NETWORK
TITLE = ---- Final
/////////////////////////////////////////////////////////////////////////
/////////////////////////////////////////////////////////////////////////
/////////////////////////////////////////////////////////////////////////
// Se acabo el evento
Final_EventoRecibido_RETI:NOP   0;
      L     #P_Eventos;  // Recupero por donde voy en la lista de eventos
      LAR2;  // Regreso a buscar el siguiente evento
      JU    FinBucle_EventosRecibidos;



NETWORK
TITLE = Guardar Datos - Evento BORR - Borrar la UT
// Analisis del evento
//   - Inicializa variables de los atributos del Evento
//   - Buscar Atributos o Final del Evento
//   - Guardar datos del Evento
// Analisis de los atributos del Evento
//   - Mirar que atributo del Evento es
//   - Distribuir a recoger los datos del Evento
//   - Recoger el Atributo McKey
//   - Recoger el Atributo MesaActual
GuardarDatos_EventoRecibido_BORR:NOP   0;

/////////////////////////////////////////////////////////////////////////
/////////////////////////////////////////////////////////////////////////
/////////////////////////////////////////////////////////////////////////
// --- Guardar Datos del Evento Recibido


/////////////////////////////////////////////////////////////////////////
/////////////////////////////////////////////////////////////////////////
/////////////////////////////////////////////////////////////////////////
// --- Control de Mesa Recibida
      L     #AtributosDeUTs.MesaActual;
      L     0;
      ==I;
      JC    FinControlMesa_EventoRecibido_BORR;

      L     #AtributosDeUTs.MesaActual;  // Ver que mesa es
      L     "CTE_OffsetMesa";
      -I;
      T     #VarTempUTs.MesaActual;

      L     #VarTempUTs.MesaActual;  // Comprobar el numero de mesa
      L     1;  // No menor de 1
      <I;  // No es correcto
      JC    Final_EventoRecibido_BORR;
      L     #VarTempUTs.MesaActual;
      L     "CTE_MaxMesas";  // No mayor que el parametro
      >I;  // No es correcto
      JC    Final_EventoRecibido_BORR;

/////////////////////////////////////////////////////////////////////////
FinControlMesa_EventoRecibido_BORR:NOP   0;



NETWORK
TITLE = ---- Accion del Evento --> Distribucion
/////////////////////////////////////////////////////////////////////////
/////////////////////////////////////////////////////////////////////////
/////////////////////////////////////////////////////////////////////////
// --- Distribucion

      L     0;  // Borrar UT en Particular
      L     #AtributosDeUTs.Mckey;
      <>D;
      JC    BorrarUT_EventoRecibido_BORR;

      L     0;  // Borrar UTs de la Mesa
      L     #AtributosDeUTs.MesaActual;
      <>I;
      JC    BorrarUTsDeMesa_EventoRecibido_BORR;

/////////////////////////////////////////////////////////////////////////
// --- Defecto --> Borrar todas las UTs
      JU    BorrarTodasLasUTs_EventoRecibido_BORR;



NETWORK
TITLE = ---- Accion del Evento --> Borrar UT
/////////////////////////////////////////////////////////////////////////
/////////////////////////////////////////////////////////////////////////
/////////////////////////////////////////////////////////////////////////
// --- Borrar una UT en particular
BorrarUT_EventoRecibido_BORR:NOP   0;
      L     #AtributosDeUTs.MesaActual;
      T     #VarTempUTs.MesaActual;
      L     0;  // Comprobar si hay mesa
      ==I;
      JC    BuscarUT_BorrarUT_EventoRecibido_BORR;

      L     #AtributosDeUTs.MesaActual;  // Ver que mesa es
      L     "CTE_OffsetMesa";
      -I;
      T     #VarTempUTs.MesaActual;

      L     #VarTempUTs.MesaActual;  // Comprobar el numero de mesa
      L     1;  // No menor de 1
      <I;  // No es correcto
      JC    Final_EventoRecibido_BORR;
      L     #VarTempUTs.MesaActual;
      L     "CTE_MaxMesas";  // No mayor que el parametro
      >I;  // No es correcto
      JC    Final_EventoRecibido_BORR;

BuscarUT_BorrarUT_EventoRecibido_BORR:NOP   0;

/////////////////////////////////////////////////////////////////////////
// --- Buscar UT en la Mesa Actual o por Mckey

      CALL  "FC720_BuscarUT_EnMesa"
      ( Mckey      := #AtributosDeUTs.Mckey,
        MesaActual := #VarTempUTs.MesaActual,
        NumeroUT   := #VarTempUTs.NumeroUT
      );

      L     #VarTempUTs.NumeroUT;
      L     0;  // No existe UT
      ==I;
      JC    Final_EventoRecibido_BORR;

/////////////////////////////////////////////////////////////////////////
// --- Modificar datos
      L     131;  // 131 - Generar Evento de Borrar UT --> ALONSO(20160525)
      T     "DB812_UTs_Control".UT[#VarTempUTs.NumeroUT].EstadoEventoAGenerar;

      JU    Final_EventoRecibido_BORR;



NETWORK
TITLE = ---- Accion del Evento --> Borrar UTs de la Mesa
/////////////////////////////////////////////////////////////////////////
/////////////////////////////////////////////////////////////////////////
/////////////////////////////////////////////////////////////////////////
// ---- Borrar todas las UT's de la Mesa
BorrarUTsDeMesa_EventoRecibido_BORR:NOP   0;
      L     #AtributosDeUTs.MesaActual;  // Ver que mesa es
      L     "CTE_OffsetMesa";
      -I;
      T     #VarTempUTs.MesaActual;

      L     #VarTempUTs.MesaActual;  // Comprobar el numero de mesa
      L     1;  // No menor de 1
      <I;  // No es correcto
      JC    Final_EventoRecibido_BORR;
      L     #VarTempUTs.MesaActual;
      L     "CTE_MaxMesas";  // No mayor que el parametro
      >I;  // No es correcto
      JC    Final_EventoRecibido_BORR;

      L     "DB810_ColasMesas".Colas[#VarTempUTs.MesaActual].UT_PrimeraMesa;
      T     #VarTempUTs.NumeroUT;


/////////////////////////////////////////////////////////////////////////
/////////////////////////////////////////////////////////////////////////
/////////////////////////////////////////////////////////////////////////
// --- Recorrido de todas la UT de la Mesa
BucleBorrarUTsDeMesa_EventoRecibido_BORR:NOP   0;
      L     #VarTempUTs.NumeroUT;
      L     0;  // No hay mas UT en la Mesa
      ==I;
      JC    Final_EventoRecibido_BORR;

      L     131;  // 131 - Generar Evento de Borrar UT --> ALONSO(20160525)
      T     "DB812_UTs_Control".UT[#VarTempUTs.NumeroUT].EstadoEventoAGenerar;

      L     "DB812_UTs_Control".UT[#VarTempUTs.NumeroUT].UT_SiguienteMesa;
      T     #VarTempUTs.NumeroUT;

/////////////////////////////////////////////////////////////////////////
// Continuo recorriendo todas las UTs de la Mesa
      JU    BucleBorrarUTsDeMesa_EventoRecibido_BORR;



NETWORK
TITLE = ---- Accion del Evento --> Borrar UTs de Todas las Mesas
/////////////////////////////////////////////////////////////////////////
/////////////////////////////////////////////////////////////////////////
/////////////////////////////////////////////////////////////////////////
// Borrar todas las UT's de la Instalacion
BorrarTodasLasUTs_EventoRecibido_BORR:NOP   0;
      L     0;
      T     #IndiceMesa;


/////////////////////////////////////////////////////////////////////////
/////////////////////////////////////////////////////////////////////////
/////////////////////////////////////////////////////////////////////////
// --- Recorrido de todas las Mesas
BucleMesasBorrarTodasLasUTs_EventoRecibido_BORR:NOP   0;
      L     #IndiceMesa;
      L     1;
      +I;
      T     #IndiceMesa;

      L     #IndiceMesa;
      L     "CTE_MaxMesas";
      >I;  // No hay mas mesas en la Instalacion
      JC    Final_EventoRecibido_BORR;


/////////////////////////////////////////////////////////////////////////
// Primera UT de la Mesa

      L     "DB810_ColasMesas".Colas[#IndiceMesa].UT_PrimeraMesa;
      T     #VarTempUTs.NumeroUT;


/////////////////////////////////////////////////////////////////////////
/////////////////////////////////////////////////////////////////////////
/////////////////////////////////////////////////////////////////////////
// --- Recorrido de todas la UT de la Mesa
BucleUTsDeMesaBorrarTodasLasUTs_EventoRecibido_BORR:NOP   0;
      L     #VarTempUTs.NumeroUT;
      L     0;
      ==I;  // No hay mas UT en la Mesa
      JC    BucleMesasBorrarTodasLasUTs_EventoRecibido_BORR;

      L     131;  // 131 - Generar Evento de Borrar UT --> ALONSO(20160525)
      T     "DB812_UTs_Control".UT[#VarTempUTs.NumeroUT].EstadoEventoAGenerar;

      L     "DB812_UTs_Control".UT[#VarTempUTs.NumeroUT].UT_SiguienteMesa;
      T     #VarTempUTs.NumeroUT;

// Continuo recorriendo de las UTs de la Mesa
      JU    BucleUTsDeMesaBorrarTodasLasUTs_EventoRecibido_BORR;



NETWORK
TITLE = ---- Final
/////////////////////////////////////////////////////////////////////////
/////////////////////////////////////////////////////////////////////////
/////////////////////////////////////////////////////////////////////////
// Se acabo el evento
Final_EventoRecibido_BORR:NOP   0;
      L     #P_Eventos;  // Recupero por donde voy en la lista de eventos
      LAR2;  // Regreso a buscar el siguiente evento
      JU    FinBucle_EventosRecibidos;



NETWORK
TITLE = Guardar Datos - Evento DATA - Notificacion de Datos de la UT
// Analizar el evento
// - Inicializa variables de los atributos del Evento
// - Buscar Atributos o Final del Evento
// - Guardar datos del Evento
// Analizar atributos del Evento
// - Distribuir a recoger los datos del Evento
// - Recoger el Atributo McKey
// - Recoger el Atributo MesaActual
// - Recoger el Atributo Tipo
// - Recoger el Atributo Codigo de Barras
// - Recoger el Atributo Grupo de UT
// - Recoger el Atributo Cantidad de UT en el Grupo
// - Recoger el Atributo Orden dentro del grupo
// - Recoger el Atributo Altura
GuardarDatos_EventoRecibido_DATA:NOP   0;

/////////////////////////////////////////////////////////////////////////
/////////////////////////////////////////////////////////////////////////
/////////////////////////////////////////////////////////////////////////
// --- Guardar Datos del Evento Recibido


/////////////////////////////////////////////////////////////////////////
/////////////////////////////////////////////////////////////////////////
/////////////////////////////////////////////////////////////////////////
// --- Control de Mesa Recibida
      L     #AtributosDeUTs.MesaActual;
      L     0;
      ==I;
      JC    FinControlMesa_DATA_EventosRecibidos;

      L     #AtributosDeUTs.MesaActual;  // Ver que mesa es
      L     "CTE_OffsetMesa";
      -I;
      T     #VarTempUTs.MesaActual;

      L     #VarTempUTs.MesaActual;  // Comprobar el numero de mesa
      L     1;  // No menor de 1
      <I;  // No es correcto
      JC    Final_EventoRecibido_DATA;  // No es correcto
      L     #VarTempUTs.MesaActual;
      L     "CTE_MaxMesas";  // No meyor que el parametro
      >I;  // No es correcto
      JC    Final_EventoRecibido_DATA;

/////////////////////////////////////////////////////////////////////////
FinControlMesa_DATA_EventosRecibidos:NOP   0;


/////////////////////////////////////////////////////////////////////////
/////////////////////////////////////////////////////////////////////////
/////////////////////////////////////////////////////////////////////////
// ---  Buscar UT, para guardar datos
      CALL  "FC720_BuscarUT_EnMesa"
      ( Mckey      := #AtributosDeUTs.Mckey,
        MesaActual := #VarTempUTs.MesaActual,
        NumeroUT   := #VarTempUTs.NumeroUT
      );

      L     #VarTempUTs.NumeroUT;
      L     0;
      ==I;  // No existe UT, no se hace por ahora
      JC    Final_EventoRecibido_DATA;



NETWORK
TITLE = ----
/////////////////////////////////////////////////////////////////////////
/////////////////////////////////////////////////////////////////////////
/////////////////////////////////////////////////////////////////////////
// --- Avisar de Evento Recibido

      L     204;  // 204 - Recibido Evento de Datos Nuevos de la UT
      T     "DB812_UTs_Control".UT[#VarTempUTs.NumeroUT].EstadoEventoRecibido;


/////////////////////////////////////////////////////////////////////////
/////////////////////////////////////////////////////////////////////////
/////////////////////////////////////////////////////////////////////////
// --- Guardar los datos de TipoCarga
      L     #AtributosDeUTs.TipoCarga;
      L     0;
      ==I;  // No hay que Cambiar el Tipo de Paleta ?
      JC    SinDatosTipoCarga_EventoRecibido_DATA;

      L     #AtributosDeUTs.TipoCarga;
      T     "DB812_UTs_Control".UT[#VarTempUTs.NumeroUT].TipoCarga;

      SET;
      R     "DB812_UTs_Control".UT[#VarTempUTs.NumeroUT].AtributosDelaCarga.Pila;
      R     "DB812_UTs_Control".UT[#VarTempUTs.NumeroUT].AtributosDelaCarga.Remontada;
      R     "DB812_UTs_Control".UT[#VarTempUTs.NumeroUT].AtributosDelaCarga.Vacia;

      SET;
      A     #AtributosDeUTs.AtributosTipoDeCarga.Pila;
      S     "DB812_UTs_Control".UT[#VarTempUTs.NumeroUT].AtributosDelaCarga.Pila;
      SET;
      A     #AtributosDeUTs.AtributosTipoDeCarga.Remontada;
      S     "DB812_UTs_Control".UT[#VarTempUTs.NumeroUT].AtributosDelaCarga.Remontada;
      SET;
      A     #AtributosDeUTs.AtributosTipoDeCarga.Vacia;
      S     "DB812_UTs_Control".UT[#VarTempUTs.NumeroUT].AtributosDelaCarga.Vacia;
SinDatosTipoCarga_EventoRecibido_DATA:NOP   0;


//////////////////////////////////////////////////////////////////////
//////////////////////////////////////////////////////////////////////
//////////////////////////////////////////////////////////////////////
// --- Se cambia todo lo relacionado con el gálibo
      L     #AtributosDeUTs.GaliboAltura;
      L     0;
      ==I;  // No hay que Cambiar la Altura ?
      JC    SinDatosGaliboAltura_EventoRecibido_DATA;

      L     #AtributosDeUTs.GaliboAltura;
      T     "DB815_UTs_Datos".UT[#VarTempUTs.NumeroUT].GaliboAltura;
SinDatosGaliboAltura_EventoRecibido_DATA:NOP   0;

//////////////////////////////////////////////////////////////////////
      L     #AtributosDeUTs.GaliboAnchura;
      L     0;
      ==I;  // No hay que Cambiar la Anchura ?
      JC    SinDatosGaliboAnchura_EventoRecibido_DATA;

      L     #AtributosDeUTs.GaliboAnchura;
      T     "DB815_UTs_Datos".UT[#VarTempUTs.NumeroUT].GaliboAnchura;
SinDatosGaliboAnchura_EventoRecibido_DATA:NOP   0;

//////////////////////////////////////////////////////////////////////
      L     #AtributosDeUTs.GaliboProfundidad;
      L     0;
      ==I;  // No hay que Cambiar la Profundidad ?
      JC    SinDatosGaliboProfundidad_EventoRecibido_DATA;

      L     #AtributosDeUTs.GaliboProfundidad;
      T     "DB815_UTs_Datos".UT[#VarTempUTs.NumeroUT].GaliboProfundidad;
SinDatosGaliboProfundidad_EventoRecibido_DATA:NOP   0;

//////////////////////////////////////////////////////////////////////
      L     #AtributosDeUTs.GaliboHueco;
      L     0;
      ==I;  // No hay que Cambiar la Hueco ?
      JC    SinDatosGaliboHueco_EventoRecibido_DATA;

      L     #AtributosDeUTs.GaliboHueco;
      T     "DB815_UTs_Datos".UT[#VarTempUTs.NumeroUT].GaliboHueco;
SinDatosGaliboHueco_EventoRecibido_DATA:NOP   0;

//////////////////////////////////////////////////////////////////////
      L     #AtributosDeUTs.GaliboTaco;
      L     0;
      ==I;  // No hay que Cambiar la Taco ?
      JC    SinDatosGaliboTaco_EventoRecibido_DATA;

      L     #AtributosDeUTs.GaliboTaco;
      T     "DB815_UTs_Datos".UT[#VarTempUTs.NumeroUT].GaliboTaco;
SinDatosGaliboTaco_EventoRecibido_DATA:NOP   0;

//////////////////////////////////////////////////////////////////////
      L     #AtributosDeUTs.GaliboHuecoRemontada;
      L     0;
      ==I;  // No hay que Cambiar la Hueco Remontada ?
      JC    SinDatosGaliboHuecoRemontada_EventoRecibido_DATA;

      L     #AtributosDeUTs.GaliboHuecoRemontada;
      T     "DB815_UTs_Datos".UT[#VarTempUTs.NumeroUT].GaliboHuecoRemontado;
SinDatosGaliboHuecoRemontada_EventoRecibido_DATA:NOP   0;


//////////////////////////////////////////////////////////////////////
      L     #AtributosDeUTs.GaliboColor;
      L     0;
      ==I;  // No hay que Cambiar la Color ?
      JC    SinDatosGaliboColor_EventoRecibido_DATA;

      L     #AtributosDeUTs.GaliboHuecoRemontada;
      T     "DB815_UTs_Datos".UT[#VarTempUTs.NumeroUT].GaliboColor;
SinDatosGaliboColor_EventoRecibido_DATA:NOP   0;

//////////////////////////////////////////////////////////////////////
      L     #AtributosDeUTs.GaliboPatin;
      L     0;
      ==I;  // No hay que Cambiar la Patin ?
      JC    SinDatosGaliboPatin_EventoRecibido_DATA;

      L     #AtributosDeUTs.GaliboPatin;
      T     "DB815_UTs_Datos".UT[#VarTempUTs.NumeroUT].GaliboPatin;
SinDatosGaliboPatin_EventoRecibido_DATA:NOP   0;







//////////////////////////////////////////////////////////////////////
      L     #AtributosDeUTs.CodigoFlejado;
      L     -1;
      ==I;  // No hay que Cambiar el Flejado ?
      JC    SinDatosCodigoFlejado_EventoRecibido_DATA;

      L     #AtributosDeUTs.CodigoFlejado;
      T     "DB815_UTs_Datos".UT[#VarTempUTs.NumeroUT].CodigoFlejado;
SinDatosCodigoFlejado_EventoRecibido_DATA:NOP   0;


//////////////////////////////////////////////////////////////////////
      L     #AtributosDeUTs.CodigoEnfardado;
      L     -1;
      ==I;  // No hay que Cambiar el Enfardado ?
      JC    SinDatosCodigoEnfardado_EventoRecibido_DATA;

      L     #AtributosDeUTs.CodigoEnfardado;
      T     "DB815_UTs_Datos".UT[#VarTempUTs.NumeroUT].CodigoEnfardado;
SinDatosCodigoEnfardado_EventoRecibido_DATA:NOP   0;


//////////////////////////////////////////////////////////////////////
      L     #AtributosDeUTs.CodigoEtiquetado;
      L     -1;
      ==I;  // No hay que Cambiar el Etiquetado ?
      JC    SinDatosCodigoEtiquetado_EventoRecibido_DATA;

      L     #AtributosDeUTs.CodigoEtiquetado;
      T     "DB815_UTs_Datos".UT[#VarTempUTs.NumeroUT].CodigoEtiquetado;
SinDatosCodigoEtiquetado_EventoRecibido_DATA:NOP   0;


//////////////////////////////////////////////////////////////////////
      L     #AtributosDeUTs.Peso;
      L     0;
      ==I;  // No hay que Cambiar el Peso ?
      JC    SinDatosPeso_EventoRecibido_DATA;

      L     #AtributosDeUTs.Peso;
      T     "DB815_UTs_Datos".UT[#VarTempUTs.NumeroUT].Peso;
SinDatosPeso_EventoRecibido_DATA:NOP   0;


//////////////////////////////////////////////////////////////////////
      L     #AtributosDeUTs.CotaAltura;
      L     0;
      ==I;  // No hay que Cambiar el Altura (Cota) ?
      JC    SinDatosCotaAltura_EventoRecibido_DATA;

      L     #AtributosDeUTs.CotaAltura;
      T     "DB815_UTs_Datos".UT[#VarTempUTs.NumeroUT].CotaAltura;
SinDatosCotaAltura_EventoRecibido_DATA:NOP   0;


//////////////////////////////////////////////////////////////////////
      L     #AtributosDeUTs.CotaAnchura;
      L     0;
      ==I;  // No hay que Cambiar el Cota Anchura ?
      JC    SinDatosCotaAnchura_EventoRecibido_DATA;

      L     #AtributosDeUTs.CotaAnchura;
      T     "DB815_UTs_Datos".UT[#VarTempUTs.NumeroUT].CotaAnchura;
SinDatosCotaAnchura_EventoRecibido_DATA:NOP   0;


//////////////////////////////////////////////////////////////////////
      L     #AtributosDeUTs.CotaProfundidad;
      L     0;
      ==I;  // No hay que Cambiar el Cota Largura ?
      JC    SinDatosCotaProfundidad_EventoRecibido_DATA;

      L     #AtributosDeUTs.CotaProfundidad;
      T     "DB815_UTs_Datos".UT[#VarTempUTs.NumeroUT].CotaProfundidad;
SinDatosCotaProfundidad_EventoRecibido_DATA:NOP   0;


//////////////////////////////////////////////////////////////////////
      L     #AtributosDeUTs.CotaAmarre;
      L     0;
      ==I;  // No hay que Cambiar el Amarre ?
      JC    SinDatosCotaAmarre_EventoRecibido_DATA;

      L     #AtributosDeUTs.CotaAmarre;
      T     "DB815_UTs_Datos".UT[#VarTempUTs.NumeroUT].Amarre;
SinDatosCotaAmarre_EventoRecibido_DATA:NOP   0;


//////////////////////////////////////////////////////////////////////
      L     #AtributosDeUTs.Presion;
      L     0;
      ==I;  // No hay que Cambiar el Presion ?
      JC    SinDatosPresion_EventoRecibido_DATA;

      L     #AtributosDeUTs.Presion;
      T     "DB815_UTs_Datos".UT[#VarTempUTs.NumeroUT].Presion;
SinDatosPresion_EventoRecibido_DATA:NOP   0;


//////////////////////////////////////////////////////////////////////
//////////////////////////////////////////////////////////////////////
//////////////////////////////////////////////////////////////////////
// --- Guardar Grupo
      L     #AtributosDeUTs.Grupo;
      L     0;
      ==I;  // No hay que Cambiar el Grupo ?
      JC    SinDatosGrupo_EventoRecibido_DATA;

      L     #AtributosDeUTs.Grupo;
      T     "DB812_UTs_Control".UT[#VarTempUTs.NumeroUT].Grupo;
      L     #AtributosDeUTs.CantidadGrupo;
      T     "DB812_UTs_Control".UT[#VarTempUTs.NumeroUT].CantidadGrupo;
      L     #AtributosDeUTs.PosicionGrupo;
      T     "DB812_UTs_Control".UT[#VarTempUTs.NumeroUT].PosicionGrupo;
SinDatosGrupo_EventoRecibido_DATA:NOP   0;


//////////////////////////////////////////////////////////////////////
//////////////////////////////////////////////////////////////////////
//////////////////////////////////////////////////////////////////////
// --- Guardar Posicion de la etiqueta

      L     #AtributosDeUTs.PosicionDeLaEtiqueta;  // Posicion de la Etiqueta
      L     1;  // Lado Derecho = 1
      ==I;
      R     "DB812_UTs_Control".UT[#VarTempUTs.NumeroUT].AtributosDeLaUT.LadoDeLaEtiqueta;

      L     #AtributosDeUTs.PosicionDeLaEtiqueta;  // Posicion de la Etiqueta
      L     2;  // Lado Izquierdo = 2
      ==I;
      S     "DB812_UTs_Control".UT[#VarTempUTs.NumeroUT].AtributosDeLaUT.LadoDeLaEtiqueta;


//////////////////////////////////////////////////////////////////////
//////////////////////////////////////////////////////////////////////
//////////////////////////////////////////////////////////////////////
// --- Guardar la Etiqueta

      L     0;
      L     #AtributosDeUTs.Etiqueta[0];
      ==I;
      JC    SinDatosEtiqueta_EventoRecibido_DATA;

      CALL  BLKMOV
      ( SRCBLK  := #AtributosDeUTs.Etiqueta,
        RET_VAL := #ReturnValor,
        DSTBLK  := "DB814_UTs_Etiqueta".UT[#VarTempUTs.NumeroUT].Etiqueta
      );
SinDatosEtiqueta_EventoRecibido_DATA:NOP   0;


//////////////////////////////////////////////////////////////////////
//////////////////////////////////////////////////////////////////////
//////////////////////////////////////////////////////////////////////
// --- Guardar Datos de QUBIQA
      L     0;
      L     #AtributosDeUTs.QUBIQA_NumeroBulto;
      ==I;
      JC    SinDatosQUBIQA_EventoRecibido_DATA;

      L     #AtributosDeUTs.QUBIQA_NumeroBulto;  // Numero de Bulto
      T     "DB820_UTs_DatosQUBIQA".UT[#VarTempUTs.NumeroUT].NumeroDeBulto;
      L     #AtributosDeUTs.QUBIQA_TotalBultos;  // Numero de Bultos
      T     "DB820_UTs_DatosQUBIQA".UT[#VarTempUTs.NumeroUT].TotalBultos;

      CALL  BLKMOV
      ( SRCBLK  := #AtributosDeUTs.QUBIQA_PID,
        RET_VAL := #ReturnValor,
        DSTBLK  := "DB820_UTs_DatosQUBIQA".UT[#VarTempUTs.NumeroUT].PID
      );  // Guardar el PID

SinDatosQUBIQA_EventoRecibido_DATA:NOP   0;



NETWORK
TITLE = ---- Final
//////////////////////////////////////////////////////////////////////
//////////////////////////////////////////////////////////////////////
//////////////////////////////////////////////////////////////////////
// Se acabo el evento
Final_EventoRecibido_DATA:NOP   0;
      L     #P_Eventos;  // Recupero por donde voy en la lista de eventos
      LAR2;
      JU    FinBucle_EventosRecibidos;  // Regreso a buscar el siguiente evento



NETWORK
TITLE = Guardar Datos - Evento ?UT? - Peticion de Refresco de datos de las UT's
// Analisis del Evento
// - Inicializa variables de los atributos del Evento
// - Buscar Atributos o Final del Evento
// - Guardar datos del Evento
//   - Si es UT determinada
//   - Si es una mesa determinada
//   - Si son todas
// Analisis de los atributos del Evento
// - Mirar que atributo del Evento es
// - Distribuir a recoger los datos del Evento
// - Recoger el Atributo McKey
// - Recoger el Atributo MesaActual
GuardarDatos_EventoRecibido_Refresco_UT:NOP   0;

/////////////////////////////////////////////////////////////////////////
/////////////////////////////////////////////////////////////////////////
/////////////////////////////////////////////////////////////////////////
// --- Guardar Datos del Evento Recibido


/////////////////////////////////////////////////////////////////////////
/////////////////////////////////////////////////////////////////////////
/////////////////////////////////////////////////////////////////////////
// --- Control de la Mesa Recibida
      L     #AtributosDeUTs.MesaActual;  // Si ha llegado atributo de Mesa
      L     0;  // Antes de comprobar si es el correcto
      ==I;  // No ha llegado
      JC    FinControlMesa_RefrescoUT_EventosRecibidos;

      L     #AtributosDeUTs.MesaActual;  // Ver que mesa es
      L     "CTE_OffsetMesa";
      -I;
      T     #VarTempUTs.MesaActual;

      L     #VarTempUTs.MesaActual;  // Comprobar el numero de mesa
      L     1;  // No menor de 1
      <I;  // No es correcto
      JC    Final_EventoRecibido_RefrescoUT;
      L     #VarTempUTs.MesaActual;
      L     "CTE_MaxMesas";  // No meyor que el parametro
      >I;  // No es correcto
      JC    Final_EventoRecibido_RefrescoUT;

/////////////////////////////////////////////////////////////////////////
FinControlMesa_RefrescoUT_EventosRecibidos:NOP   0;



NETWORK
TITLE = ---- Accion del Evento --> Distribucion
/////////////////////////////////////////////////////////////////////////
/////////////////////////////////////////////////////////////////////////
/////////////////////////////////////////////////////////////////////////
// --- Distribucion para la busqueda

      L     #AtributosDeUTs.Mckey;
      L     0;
      <>I;  // Es una UT Especifica
      JC    RefrescoDeUT_EventoRecibido_RefrescoUT;

      L     #AtributosDeUTs.MesaActual;
      L     0;
      <>I;  // Son todas las UT de una Mesa
      JC    RefrescoDeUTsDeLaMesa_EventoRecibido_RefrescoUT;

/////////////////////////////////////////////////////////////////////////
// --- Son todas las UT -> Por defecto
      JU    RefrescoDeUTsTodasLasMesas_EventoRecibido_RefrescoUT;



NETWORK
TITLE = ---- Accion del Evento --> Peticion de Refesco de una UT especifica
/////////////////////////////////////////////////////////////////////////
/////////////////////////////////////////////////////////////////////////
/////////////////////////////////////////////////////////////////////////
// Es una UT Especifica
RefrescoDeUT_EventoRecibido_RefrescoUT:NOP   0;
      L     #AtributosDeUTs.MesaActual;
      T     #VarTempUTs.MesaActual;
      L     0;  // Comprobar si hay mesa
      ==I;
      JC    BuscarUT_RefrescoDeUT_EventoRecibido_RefrescoUT;

      L     #AtributosDeUTs.MesaActual;  // Ver que mesa es
      L     "CTE_OffsetMesa";
      -I;
      T     #VarTempUTs.MesaActual;

      L     #VarTempUTs.MesaActual;  // Comprobar el numero de mesa
      L     1;  // No menor de 1
      <I;  // No es correcto
      JC    Final_EventoRecibido_RefrescoUT;
      L     #VarTempUTs.MesaActual;
      L     "CTE_MaxMesas";  // No mayor que el parametro
      >I;  // No es correcto
      JC    Final_EventoRecibido_RefrescoUT;

BuscarUT_RefrescoDeUT_EventoRecibido_RefrescoUT:NOP   0;
      CALL  "FC720_BuscarUT_EnMesa"
      ( Mckey      := #AtributosDeUTs.Mckey,
        MesaActual := #VarTempUTs.MesaActual,
        NumeroUT   := #VarTempUTs.NumeroUT  // Donde esta la UT
      );  // Busca por Mesa o por Mckey

      L     #VarTempUTs.NumeroUT;
      L     0;
      ==I;  // No existe UT, no se hace por ahora
      JC    Final_EventoRecibido_RefrescoUT;


/////////////////////////////////////////////////////////////////////////
/// Generar Peticion de Datos de la UT
// 205 - Recibido Evento de Refesco de datos para la UT (Anulado)
// 22  - Estado General UT Peticion de Refresco de datos

// 2023 01 05 - Anulado >>> Cambio de Sistema
//      L     22                   // 22 - Peticion de Refresco de datos
//      T     "DB812_UTs_Control".UT[#VarTempUTs.NumeroUT].EstadoGeneralUT
// 2023 01 05 - Bits para informar >>> Nueco Sistema
      SET;
      =     "DB812_UTs_Control".UT[#VarTempUTs.NumeroUT].EventosInformarJdT.PeticionDeDatos;

      JU    Final_EventoRecibido_RefrescoUT;



NETWORK
TITLE = ---- Accion del Evento --> Peticion de Refesco de las UTs de una Mesa
/////////////////////////////////////////////////////////////////////////
/////////////////////////////////////////////////////////////////////////
/////////////////////////////////////////////////////////////////////////
// --- Son todas las UT de una Mesa
RefrescoDeUTsDeLaMesa_EventoRecibido_RefrescoUT:NOP   0;
      L     #AtributosDeUTs.MesaActual;  // Ver que mesa es
      L     "CTE_OffsetMesa";
      -I;
      T     #VarTempUTs.MesaActual;

      L     #VarTempUTs.MesaActual;  // Comprobar el numero de mesa
      L     1;  // No menor de 1
      <I;  // No es correcto
      JC    Final_EventoRecibido_RefrescoUT;
      L     #VarTempUTs.MesaActual;
      L     "CTE_MaxMesas";  // No mayor que el parametro
      >I;  // No es correcto
      JC    Final_EventoRecibido_RefrescoUT;

/////////////////////////////////////////////////////////////////////////
/// --- Mirar si esta definido como mesa de tracking
      SET;
      AN    "DB850_DefinicionMesas".Mesa[#VarTempUTs.MesaActual].ConfigMesa.MesaPaso;
      AN    "DB850_DefinicionMesas".Mesa[#VarTempUTs.MesaActual].ConfigMesa.MesaCruce;
      AN    "DB850_DefinicionMesas".Mesa[#VarTempUTs.MesaActual].ConfigMesa.MesaMultiplesDestinos;
      JC    Final_EventoRecibido_RefrescoUT;


/////////////////////////////////////////////////////////////////////////
/// --- Mirar Si pertenece al JDT // JDT01 ?
      SET;
      X     "DB850_DefinicionMesas".Mesa[#VarTempUTs.MesaActual].ConfigMesa.MesaDeJDT02;
      XN    #JDT02_Activo;
      =     #MesaDeJDT02;

      SET;
      AN    #MesaDeJDT02;
      JC    Final_EventoRecibido_RefrescoUT;


/////////////////////////////////////////////////////////////////////////
// --- Primera UT de la Mesa
      L     "DB810_ColasMesas".Colas[#VarTempUTs.MesaActual].UT_PrimeraMesa;
      T     #VarTempUTs.NumeroUT;


/////////////////////////////////////////////////////////////////////////
/////////////////////////////////////////////////////////////////////////
/////////////////////////////////////////////////////////////////////////
BucleRefrescoUTsDeMesa_EventoRecibido_RefrescoUT:NOP   0;
      L     #VarTempUTs.NumeroUT;  // Recorrido de todas la UT de la Mesa
      L     0;
      ==I;  // No hay mas UT en la Mesa
      JC    Final_EventoRecibido_RefrescoUT;

/////////////////////////////////////////////////////////////////////////
/// Generar Peticion de Datos de la UT
// 205 - Recibido Evento de Refesco de datos para la UT (Anulado)
// 22  - Estado General UT Peticion de Refresco de datos

// 2023 01 05 - Anulado >>> Cambio de Sistema
//      L     22                   // 22 - Peticion de Refresco de datos
//      T     "DB812_UTs_Control".UT[#VarTempUTs.NumeroUT].EstadoGeneralUT
// 2023 01 05 - Bits para informar >>> Nueco Sistema
      SET;
      =     "DB812_UTs_Control".UT[#VarTempUTs.NumeroUT].EventosInformarJdT.PeticionDeDatos;

/////////////////////////////////////////////////////////////////////////
// --- Continuo recorriendo la Mesa
      L     "DB812_UTs_Control".UT[#VarTempUTs.NumeroUT].UT_SiguienteMesa;
      T     #VarTempUTs.NumeroUT;
      JU    BucleRefrescoUTsDeMesa_EventoRecibido_RefrescoUT;



NETWORK
TITLE = ---- Accion del Evento --> Peticion de Refesco de las UTs de Todas las Mesas
/////////////////////////////////////////////////////////////////////////
/////////////////////////////////////////////////////////////////////////
/////////////////////////////////////////////////////////////////////////
// --- Son todas las UT de la Instalacion
RefrescoDeUTsTodasLasMesas_EventoRecibido_RefrescoUT:NOP   0;

      L     0;
      T     #IndiceMesa;

/////////////////////////////////////////////////////////////////////////
/////////////////////////////////////////////////////////////////////////
/////////////////////////////////////////////////////////////////////////
// --- Recorrido de todas las Mesas
BucleMesaRefrescoUTsDeMesa_EventoRecibido_RefrescoUT:NOP   0;
      L     #IndiceMesa;
      L     1;
      +I;
      T     #IndiceMesa;

      L     #IndiceMesa;
      L     "CTE_MaxMesas";
      >I;  // No hay mas mesas en la Instalacion
      JC    Final_EventoRecibido_RefrescoUT;


/////////////////////////////////////////////////////////////////////////
/// --- Mirar si esta definido como mesa de tracking
      SET;
      AN    "DB850_DefinicionMesas".Mesa[#IndiceMesa].ConfigMesa.MesaPaso;
      AN    "DB850_DefinicionMesas".Mesa[#IndiceMesa].ConfigMesa.MesaCruce;
      AN    "DB850_DefinicionMesas".Mesa[#IndiceMesa].ConfigMesa.MesaMultiplesDestinos;
      JC    BucleMesaRefrescoUTsDeMesa_EventoRecibido_RefrescoUT;


/////////////////////////////////////////////////////////////////////////
/// --- Mirar Si pertenece al JDT
      SET;
      X     "DB850_DefinicionMesas".Mesa[#IndiceMesa].ConfigMesa.MesaDeJDT02;  // JDT01 ?
      XN    #JDT02_Activo;
      =     #MesaDeJDT02;

      SET;
      AN    #MesaDeJDT02;
      JC    BucleMesaRefrescoUTsDeMesa_EventoRecibido_RefrescoUT;


/////////////////////////////////////////////////////////////////////////
/////////////////////////////////////////////////////////////////////////
/////////////////////////////////////////////////////////////////////////
// --- Recorrer la Mesa

      L     "DB810_ColasMesas".Colas[#IndiceMesa].UT_PrimeraMesa;
      T     #VarTempUTs.NumeroUT;

BucleUTsMesaRefrescoUTsDeMesa_EventoRecibido_RefrescoUT:NOP   0;
      L     #VarTempUTs.NumeroUT;  // Recorrido de todas la UT de la Mesa
      L     0;
      ==I;  // No hay mas UT en la Mesa
      JC    BucleMesaRefrescoUTsDeMesa_EventoRecibido_RefrescoUT;

/////////////////////////////////////////////////////////////////////////
/// --- Generar Peticion de Datos de la UT
// 205 - Recibido Evento de Refesco de datos para la UT (Anulado)
// 22  - Estado General UT Peticion de Refresco de datos

// 2023 01 05 - Anulado >>> Cambio de Sistema
//      L     22                   // 22 - Peticion de Refresco de datos
//      T     "DB812_UTs_Control".UT[#VarTempUTs.NumeroUT].EstadoGeneralUT
// 2023 01 05 - Bits para informar >>> Nueco Sistema
      SET;
      =     "DB812_UTs_Control".UT[#VarTempUTs.NumeroUT].EventosInformarJdT.PeticionDeDatos;

/////////////////////////////////////////////////////////////////////////
// --- Continuo recorriendo la Mesa
      L     "DB812_UTs_Control".UT[#VarTempUTs.NumeroUT].UT_SiguienteMesa;
      T     #VarTempUTs.NumeroUT;
      JU    BucleUTsMesaRefrescoUTsDeMesa_EventoRecibido_RefrescoUT;



NETWORK
TITLE = ---- Final
////////////////////////////////////////////////////////////////////////////////////////
////////////////////////////////////////////////////////////////////////////////////////
////////////////////////////////////////////////////////////////////////////////////////
// Se acabo el evento
Final_EventoRecibido_RefrescoUT:NOP   0;
      L     #P_Eventos;  // Recupero por donde voy en la lista de eventos
      LAR2;  // Regreso a buscar el siguiente evento
      JU    FinBucle_EventosRecibidos;



NETWORK
TITLE = Guardar Datos - Evento MOVE - Mover UT de Mesa // 08 02 2017
GuardarDatos_EventoRecibido_MOVE:NOP   0;

/////////////////////////////////////////////////////////////////////////
/////////////////////////////////////////////////////////////////////////
/////////////////////////////////////////////////////////////////////////
// --- Guardar Datos del Evento Recibido


/////////////////////////////////////////////////////////////////////////
/////////////////////////////////////////////////////////////////////////
/////////////////////////////////////////////////////////////////////////
// --- Control de Mesa Recibida
      L     #AtributosDeUTs.MesaActual;  // Ver que mesa es
      L     "CTE_OffsetMesa";
      -I;
      T     #VarTempUTs.MesaActual;

      L     #VarTempUTs.MesaActual;  // Comprobar el numero de mesa
      L     1;  // No menor de 1
      <I;  // No es correcto
      JC    Final_EventoRecibido_MOVE;
      L     #VarTempUTs.MesaActual;
      L     "CTE_MaxMesas";  // No mayor que el parametro
      >I;  // No es correcto
      JC    Final_EventoRecibido_MOVE;


///////////////////////////////////////////////////////////////////////////////
// --- Control de McKey Recibido
      L     #AtributosDeUTs.Mckey;  // Se ha recibido Mckey = 0
      L     0;  // No se puede Crear
      ==D;
      JC    Final_EventoRecibido_MOVE;


///////////////////////////////////////////////////////////////////////////////
// --- Busca el Mckey Recibido, comprobar que existe

      CALL  "FC720_BuscarUT_EnMesa"
      ( Mckey      := #AtributosDeUTs.Mckey,
        MesaActual := #VarTempUTs.MesaActual,
        NumeroUT   := #VarTempUTs.NumeroUT
      );

      L     #VarTempUTs.NumeroUT;
      L     0;
      ==I;  // No Existe UT ?
      JC    Final_EventoRecibido_MOVE;



NETWORK
TITLE = ---- Accion del Evento
///////////////////////////////////////////////////////////////////////////////
///////////////////////////////////////////////////////////////////////////////
///////////////////////////////////////////////////////////////////////////////
// --- Guardar Respuesta

      SET;
      L     "DB812_UTs_Control".UT[#VarTempUTs.NumeroUT].MesaActual;
      L     #AtributosDeUTs.MesaActual;
      <>I;  // Esta en Mesa diferente ?
      JC    Final_EventoRecibido_MOVE;

      SET;  // Realizada la peticion de Cambio de Mesa ?
      AN    "DB812_UTs_Control".UT[#VarTempUTs.NumeroUT].EventosDeCambioDeMesa.PeticionCambiarUTDeMesa;
      JC    Final_EventoRecibido_MOVE;


///////////////////////////////////////////////////////////////////////////////
///////////////////////////////////////////////////////////////////////////////
///////////////////////////////////////////////////////////////////////////////
// --- Orden Recibida guardarla en la UT

      SET;  // OK Cambiar UT de Mesa Final
      A     #AtributosDeUTs.CambiarUTDeMesa.OK;
      A     #AtributosDeUTs.CambiarUTDeMesa.Final;
      S     "DB812_UTs_Control".UT[#VarTempUTs.NumeroUT].EventosDeCambioDeMesa.OKCambiarUTDeMesaFinal;

      SET;  // OK Cambiar UT de Mesa Inicio
      A     #AtributosDeUTs.CambiarUTDeMesa.OK;
      A     #AtributosDeUTs.CambiarUTDeMesa.Inicio;
      S     "DB812_UTs_Control".UT[#VarTempUTs.NumeroUT].EventosDeCambioDeMesa.OKCambiarUTDeMesaInicio;

      SET;  // NOK Cambiar UT de Mesa
      A     #AtributosDeUTs.CambiarUTDeMesa.NOK;
      S     "DB812_UTs_Control".UT[#VarTempUTs.NumeroUT].EventosDeCambioDeMesa.NOKCambiarUTDeMesa;


///////////////////////////////////////////////////////////////////////////////
      JU    Final_EventoRecibido_MOVE;



NETWORK
TITLE = ---- Final
///////////////////////////////////////////////////////////////////////////////
///////////////////////////////////////////////////////////////////////////////
///////////////////////////////////////////////////////////////////////////////
// Se acabo el evento
Final_EventoRecibido_MOVE:NOP   0;
      L     #P_Eventos;  // Recupero por donde voy en la lista de eventos
      LAR2;
      JU    FinBucle_EventosRecibidos;



NETWORK
TITLE = Guardar Datos - Evento DEMB - Datos de EmBandejado de la UT // Fecha 07 06 2017
GuardarDatos_EventoRecibido_DEMB:NOP   0;

/////////////////////////////////////////////////////////////////////////
/////////////////////////////////////////////////////////////////////////
/////////////////////////////////////////////////////////////////////////
// --- Guardar Datos del Evento Recibido


/////////////////////////////////////////////////////////////////////////
/////////////////////////////////////////////////////////////////////////
/////////////////////////////////////////////////////////////////////////
// --- Control de Mesa Recibida
      L     #AtributosDeUTs.MesaActual;
      L     0;
      ==I;
      JC    FinControlMesa_EventoRecibido_DEMB;

      L     #AtributosDeUTs.MesaActual;  // Ver que mesa es
      L     "CTE_OffsetMesa";
      -I;
      T     #VarTempUTs.MesaActual;

      L     #VarTempUTs.MesaActual;  // Comprobar el numero de mesa
      L     1;  // No menor de 1
      <I;  // No es correcto
      JC    Final_EventoRecibido_DEMB;
      L     #VarTempUTs.MesaActual;
      L     "CTE_MaxMesas";  // No mayor que el parametro
      >I;  // No es correcto
      JC    Final_EventoRecibido_DEMB;

/////////////////////////////////////////////////////////////////////////
FinControlMesa_EventoRecibido_DEMB:NOP   0;


/////////////////////////////////////////////////////////////////////////
/////////////////////////////////////////////////////////////////////////
/////////////////////////////////////////////////////////////////////////
// --- Control de Mckey Recibido
      L     #AtributosDeUTs.Mckey;  // Se ha recibido Mckey = 0
      L     0;  // No se puede Crear
      ==D;
      JC    Final_EventoRecibido_DEMB;


/////////////////////////////////////////////////////////////////////////
/////////////////////////////////////////////////////////////////////////
/////////////////////////////////////////////////////////////////////////
// --- Comprobar que Existe una UT
      CALL  "FC720_BuscarUT_EnMesa"
      ( Mckey      := #AtributosDeUTs.Mckey,
        MesaActual := #VarTempUTs.MesaActual,
        NumeroUT   := #VarTempUTs.NumeroUT
      );

      L     #VarTempUTs.NumeroUT;
      L     0;
      ==I;  // No Existe UT ?
      JC    Final_EventoRecibido_DEMB;



NETWORK
TITLE = ---- Accion del Evento
/////////////////////////////////////////////////////////////////////////
/////////////////////////////////////////////////////////////////////////
/////////////////////////////////////////////////////////////////////////
// Guardar Respuesta


      L     #AtributosDeUTs.QUBIQA_NumeroBulto;  // Numero de Bulto
      T     "DB820_UTs_DatosQUBIQA".UT[#VarTempUTs.NumeroUT].NumeroDeBulto;
      L     #AtributosDeUTs.QUBIQA_TotalBultos;  // Numero de Bultos
      T     "DB820_UTs_DatosQUBIQA".UT[#VarTempUTs.NumeroUT].TotalBultos;

      CALL  BLKMOV
      ( SRCBLK  := #AtributosDeUTs.QUBIQA_PID,
        RET_VAL := #ReturnValor,
        DSTBLK  := "DB820_UTs_DatosQUBIQA".UT[#VarTempUTs.NumeroUT].PID
      );  // Guardar el PID

      JU    Final_EventoRecibido_DEMB;



NETWORK
TITLE = ---- Final
/////////////////////////////////////////////////////////////////////////
/////////////////////////////////////////////////////////////////////////
/////////////////////////////////////////////////////////////////////////
// Se acabo el evento
Final_EventoRecibido_DEMB:NOP   0;
      L     #P_Eventos;  // Recupero por donde voy en la lista de eventos
      LAR2;
      JU    FinBucle_EventosRecibidos;



NETWORK
TITLE = ////////////////////////////////////////////////////////////////////////////////////////////////////////////

NETWORK
TITLE = Evento CSTA - Notificacion de cambio de Estado de un dispositivo
// Analisis del evento
// - Inicializa variables de los atributos del Evento
// - Buscar Atributos o Final del Evento
// - Guardar datos del Evento
//   - Si es tipo CCPIF (50)
//   - Si es tipo CBOX (40)
//   - Si es tipo Mesa (60)
//   - Si es tipo Maquina (70)
// Analisis de los atributos de los eventos
// - Mirar que atributo del Evento es ?
// - Distribuir a recoger los datos del Evento
// - Recoger el Atributo Tipo de Dispositivo
// - Recoger el Atributo Numero de Dispositivo
// - Recoger el Atributo Nuevo Estado del Dispositivo
GuardarDatos_EventoRecibido_CSTA:NOP   0;

/////////////////////////////////////////////////////////////////////////
/////////////////////////////////////////////////////////////////////////
/////////////////////////////////////////////////////////////////////////
// --- Guardar Datos del Evento Recibido


/////////////////////////////////////////////////////////////////////////
/////////////////////////////////////////////////////////////////////////
/////////////////////////////////////////////////////////////////////////
// --- Repartir segun tipo de dispositivo: CCPIF, CBOX, Mesa ....

      SET;  // Es CCPIF
      L     #AtributosDeDispositivos.Tipo;
      L     50;
      ==I;
      JC    DispositivosCCPIF_EventoRecibido_CSTA;

      SET;  // Es CBOX
      L     #AtributosDeDispositivos.Tipo;
      L     40;
      ==I;
      JC    DispositivosCBOX_EventoRecibido_CSTA;

      SET;  // Es Mesa
      L     #AtributosDeDispositivos.Tipo;
      L     60;
      ==I;
      JC    DispositivosMesa_EventoRecibido_CSTA;

      SET;  // Es Baliza
      L     #AtributosDeDispositivos.Tipo;
      L     1000;
      ==I;
      JC    DispositivosBaliza_EventoRecibido_CSTA;

/////////////////////////////////////////////////////////////////////////
/////////////////////////////////////////////////////////////////////////
/////////////////////////////////////////////////////////////////////////

      SET;  // Es Llave
      L     #AtributosDeDispositivos.Tipo;
      L     1001;
      ==I;
      JC    DispositivosLlave_EventoRecibido_CSTA;

      SET;  // Es Seta
      L     #AtributosDeDispositivos.Tipo;
      L     1002;
      ==I;
      JC    DispositivosSeta_EventoRecibido_CSTA;

      SET;  // Es Barrera
      L     #AtributosDeDispositivos.Tipo;
      L     1003;
      ==I;
      JC    DispositivosBarrera_EventoRecibido_CSTA;

      SET;  // Es Puerta
      L     #AtributosDeDispositivos.Tipo;
      L     1004;
      ==I;
      JC    DispositivosPuerta_EventoRecibido_CSTA;

      SET;  // Es Linea de Potencia
      L     #AtributosDeDispositivos.Tipo;
      L     1005;
      ==I;
      JC    DispositivosLineaPotencia_EventoRecibido_CSTA;


/////////////////////////////////////////////////////////////////////////
/////////////////////////////////////////////////////////////////////////
/////////////////////////////////////////////////////////////////////////
// Es Maquina De 70 ... 99
      SET;
      A(;
      L     #AtributosDeDispositivos.Tipo;
      L     70;
      >=I;
      );
      A(;
      SET;
      L     #AtributosDeDispositivos.Tipo;
      L     99;
      <=I;
      );
      JC    DispositivosMaquina_EventoRecibido_CSTA;


/////////////////////////////////////////////////////////////////////////
/////////////////////////////////////////////////////////////////////////
/////////////////////////////////////////////////////////////////////////
// --- No es ningun Tipo de Dispositivo Esperado
      JU    Final_EventoRecibido_CSTA;



NETWORK
TITLE = ---- Accion del Evento --> Notificacion de cambio de Estado de CCPIF
///////////////////////////////////////////////////////////////////////////////
///////////////////////////////////////////////////////////////////////////////
///////////////////////////////////////////////////////////////////////////////
// --- Tipo CCPIF
DispositivosCCPIF_EventoRecibido_CSTA:NOP   0;


///////////////////////////////////////////////////////////////////////////////
// --- Comprobacion del Numero de Dispositivo
      L     #AtributosDeDispositivos.Numero;  // Comprobacion del numero de CCPIF
      L     "CTE_OffsetCCPIF";
      -I;
      L     1;
      <>I;  // Numero de CCPIF incorrecto
      JC    Final_EventoRecibido_CSTA;


///////////////////////////////////////////////////////////////////////////////
// --- Guardar el Cambio de Estado Recibido
      L     #AtributosDeDispositivos.NuevoEstado;  // EstadoDispo + 260 = Recibido Evento de Cambio de Estado
      L     260;  // Orden a guardar en el DB
      +I;
      T     "DB830_Dispositivos".Dispositivos[0].EstadoRecepcionEvento;


///////////////////////////////////////////////////////////////////////////////
// --- Finalizar
      JU    Final_EventoRecibido_CSTA;



NETWORK
TITLE = ---- Accion del Evento --> Notificacion de cambio de Estado de CBOX
///////////////////////////////////////////////////////////////////////////////
///////////////////////////////////////////////////////////////////////////////
///////////////////////////////////////////////////////////////////////////////
// --- Tipo CBOX
DispositivosCBOX_EventoRecibido_CSTA:NOP   0;


///////////////////////////////////////////////////////////////////////////////
// --- Comprobacion del Numero de Dispositivo
      L     #AtributosDeDispositivos.Numero;  // Comprobacion del numero de CCPIF
      L     100;
      /I;
      L     "CTE_OffsetCCPIF";
      -I;
      L     1;
      <>I;  // Numero de CCPIF incorrecto
      JC    Final_EventoRecibido_CSTA;


      L     #AtributosDeDispositivos.Numero;  // Calculo del numero de CBOX
      L     100;
      MOD;  // Var verlo en la DB_Dispositivos
      T     #VarTempDispositivos.Numero;

      L     #VarTempDispositivos.Numero;  // Comprobacion del numero de CBOX
      L     1;  // Es menor de 1
      <I;  // No es correcto el numero de CBOX
      JC    Final_EventoRecibido_CSTA;
      L     #VarTempDispositivos.Numero;
      L     "CTE_MaxDispositivos";  // Si es mayor que el parametro
      >I;  // No es correcto el numero de CBOX
      JC    Final_EventoRecibido_CSTA;


///////////////////////////////////////////////////////////////////////////////
// --- Guardar el Cambio de Estado Recibido
      L     #AtributosDeDispositivos.NuevoEstado;  // EstadoDispo + 260 = Recibido Evento de Cambio de Estado
      L     260;  // Orden a guardar en el DB
      +I;
      T     "DB830_Dispositivos".Dispositivos[#VarTempDispositivos.Numero].EstadoRecepcionEvento;


///////////////////////////////////////////////////////////////////////////////
// --- Finalizar
      JU    Final_EventoRecibido_CSTA;



NETWORK
TITLE = ---- Accion del Evento --> Notificacion de cambio de Estado de Mesa
///////////////////////////////////////////////////////////////////////////////
///////////////////////////////////////////////////////////////////////////////
///////////////////////////////////////////////////////////////////////////////
// --- Tipo Mesa
DispositivosMesa_EventoRecibido_CSTA:NOP   0;


///////////////////////////////////////////////////////////////////////////////
// --- Comprobacion del Numero de Dispositivo
      L     #AtributosDeDispositivos.Numero;  // Ver que mesa es
      L     "CTE_OffsetMesa";
      -I;
      T     #VarTempDispositivos.Numero;

      L     #VarTempDispositivos.Numero;  // Comprobar el numero de mesa
      L     1;  // No menor de 1
      <I;  // No es correcto
      JC    Final_EventoRecibido_CSTA;
      L     #VarTempDispositivos.Numero;
      L     "CTE_MaxMesas";  // No meyor que el parametro
      >I;  // No es correcto
      JC    Final_EventoRecibido_CSTA;


///////////////////////////////////////////////////////////////////////////////
// --- Guardar el Cambio de Estado Recibido
      L     #AtributosDeDispositivos.NuevoEstado;  // EstadoDispo + 260 = Recibido Evento de Cambio de Estado
      L     260;  // Orden a guardar en el DB
      +I;
      T     "DB831_Mesas".Mesas[#VarTempDispositivos.Numero].EstadoRecepcionEvento;


///////////////////////////////////////////////////////////////////////////////
// --- Habilitado o DesHabilitado el Dispositivo
      SET;
      L     #AtributosDeDispositivos.Habilitado;
      L     2001;  // Habitar Disposito = 0
      ==I;
      R     "DB831_Mesas".Mesas[#VarTempDispositivos.Numero].Memorias.DesHabilitado;

      SET;
      L     #AtributosDeDispositivos.Habilitado;
      L     2002;  // DesHabitar Disposito = 1
      ==I;
      S     "DB831_Mesas".Mesas[#VarTempDispositivos.Numero].Memorias.DesHabilitado;


///////////////////////////////////////////////////////////////////////////////
// Prioridad  - 1...x
      SET;
      L     #AtributosDeDispositivos.Prioridad;
      L     0;
      ==I;
      JC    SinPrioridadMesa_EventoRecibido_CSTA;

      L     #AtributosDeDispositivos.Prioridad;
      T     "DB831_Mesas".Mesas[#VarTempDispositivos.Numero].Prioridad;

SinPrioridadMesa_EventoRecibido_CSTA:NOP   0;


///////////////////////////////////////////////////////////////////////////////
// --- Fecha: 08 02 2017
// --- Motivo para la pantalla del Error envio por el JDT
      SET;
      L     #LonguitudTextoRecibido;
      L     0;
      ==I;  // Existe Motivo de Error en Mesa Enviado por el JDT
      JC    SinMotivoDeErrorDelJdT_EventoRecibido_CSTA;

      CALL  BLKMOV
      ( SRCBLK  := #AtributosDeDispositivos.MotivoDelError,
        RET_VAL := #ReturnValor,
        DSTBLK  := "DB907_TextoErrorJdT".Mesa[#VarTempDispositivos.Numero]
      );

SinMotivoDeErrorDelJdT_EventoRecibido_CSTA:NOP   0;


///////////////////////////////////////////////////////////////////////////////
// --- Finalizar
      JU    Final_EventoRecibido_CSTA;



NETWORK
TITLE = ---- Accion del Evento --> Notificacion de cambio de Estado de Maquina
///////////////////////////////////////////////////////////////////////////////
///////////////////////////////////////////////////////////////////////////////
///////////////////////////////////////////////////////////////////////////////
// --- Tipo Maquina
DispositivosMaquina_EventoRecibido_CSTA:NOP   0;


///////////////////////////////////////////////////////////////////////////////
// --- Comprobacion del Numero de Dispositivo
      L     #AtributosDeDispositivos.Numero;  // Ver que mesa es
      L     "CTE_OffsetMesa";
      -I;
      T     #VarTempDispositivos.Numero;

      L     #VarTempDispositivos.Numero;  // Comprobar el numero de maquina
      L     1;  // No menor de 1
      <I;  // No es correcto
      JC    Final_EventoRecibido_CSTA;
      L     #VarTempDispositivos.Numero;
      L     "CTE_MaxMesas";  // No meyor que el parametro
      >I;  // No es correcto
      JC    Final_EventoRecibido_CSTA;


///////////////////////////////////////////////////////////////////////////////
// --- Guardar el Cambio de Estado Recibido

      L     #AtributosDeDispositivos.NuevoEstado;  // EstadoDispo + 260 = Recibido Evento de Cambio de Estado
      L     260;  // Orden a guardar en el DB
      +I;
      T     "DB832_Maquinas".Maquinas[#VarTempDispositivos.Numero].EstadoRecepcionEvento;


///////////////////////////////////////////////////////////////////////////////
// --- Habilitado o DesHabilitado
      SET;
      L     #AtributosDeDispositivos.Habilitado;
      L     2001;  // Habitar Disposito = 0
      ==I;
      R     "DB832_Maquinas".Maquinas[#VarTempDispositivos.Numero].Memorias.DesHabilitado;

      SET;
      L     #AtributosDeDispositivos.Habilitado;
      L     2002;  // DesHabitar Disposito = 1
      ==I;
      S     "DB832_Maquinas".Maquinas[#VarTempDispositivos.Numero].Memorias.DesHabilitado;


///////////////////////////////////////////////////////////////////////////////
// Prioridad  - 1...x
      SET;
      L     #AtributosDeDispositivos.Prioridad;
      L     0;
      ==I;
      JC    SinPrioridadMaquina_EventoRecibido_CSTA;

      L     #AtributosDeDispositivos.Prioridad;
      T     "DB832_Maquinas".Maquinas[#VarTempDispositivos.Numero].Prioridad;

SinPrioridadMaquina_EventoRecibido_CSTA:NOP   0;


///////////////////////////////////////////////////////////////////////////////
// Finalizar
      JU    Final_EventoRecibido_CSTA;



NETWORK
TITLE = ---- Accion del Evento --> Notificacion de cambio de Estado de Baliza
///////////////////////////////////////////////////////////////////////////////
///////////////////////////////////////////////////////////////////////////////
///////////////////////////////////////////////////////////////////////////////
// --- Tipo Baliza
DispositivosBaliza_EventoRecibido_CSTA:NOP   0;


///////////////////////////////////////////////////////////////////////////////
// --- Comprobacion del Numero de Dispositivo
      L     #AtributosDeDispositivos.Numero;  // Ver que Baliza es
      L     "CTE_OffsetMesa";
      -I;
      T     #VarTempDispositivos.Numero;

      L     #VarTempDispositivos.Numero;  // Comprobar el numero de Baliza
      L     1;  // No menor de 1
      <I;  // No es correcto
      JC    Final_EventoRecibido_CSTA;
      L     #VarTempDispositivos.Numero;
      L     "CTE_MaxDispositivosBaliza";  // No meyor que el parametro
      >I;  // No es correcto
      JC    Final_EventoRecibido_CSTA;


///////////////////////////////////////////////////////////////////////////////
// --- Guardar el Cambio de Estado Recibido

      CALL  BLKMOV
      ( SRCBLK  := "DB839_DispositivosVarios".DispoBaliza[#VarTempDispositivos.Numero],
        RET_VAL := #ReturnValor,
        DSTBLK  := #VarTempDispositivos.Baliza
      );

      SET;  // Reseteo para actualizar
      R     #VarTempDispositivos.Baliza.Sonoro;
      R     #VarTempDispositivos.Baliza.Verde;
      R     #VarTempDispositivos.Baliza.Rojo;
      R     #VarTempDispositivos.Baliza.Amarillo;
      R     #VarTempDispositivos.Baliza.Azul;


      SET;  // Sonoro
      A     #AtributosDeDispositivos.BalizaColor.Sonoro;
      S     #VarTempDispositivos.Baliza.Sonoro;

      SET;  // Verde
      A     #AtributosDeDispositivos.BalizaColor.Verde;
      S     #VarTempDispositivos.Baliza.Verde;

      SET;  // Rojo
      A     #AtributosDeDispositivos.BalizaColor.Rojo;
      S     #VarTempDispositivos.Baliza.Rojo;

      SET;  // Amarillo
      A     #AtributosDeDispositivos.BalizaColor.Amarillo;
      S     #VarTempDispositivos.Baliza.Amarillo;

      SET;  // Azul
      A     #AtributosDeDispositivos.BalizaColor.Azul;
      S     #VarTempDispositivos.Baliza.Azul;

      SET;  // Peticion de Estado
      S     #VarTempDispositivos.Baliza.RefrescoDatos;

      CALL  BLKMOV
      ( SRCBLK  := #VarTempDispositivos.Baliza,
        RET_VAL := #ReturnValor,
        DSTBLK  := "DB839_DispositivosVarios".DispoBaliza[#VarTempDispositivos.Numero]
      );


///////////////////////////////////////////////////////////////////////////////
// Finalizar
      JU    Final_EventoRecibido_CSTA;



NETWORK
TITLE = ---- Accion del Evento --> Notificacion de cambio de Estado de Llave
///////////////////////////////////////////////////////////////////////////////
///////////////////////////////////////////////////////////////////////////////
///////////////////////////////////////////////////////////////////////////////
// --- Tipo Llave
DispositivosLlave_EventoRecibido_CSTA:NOP   0;


///////////////////////////////////////////////////////////////////////////////
// --- Comprobacion del Numero de Dispositivo
      L     #AtributosDeDispositivos.Numero;  // Ver que Llave es
      L     "CTE_OffsetMesa";
      -I;
      T     #VarTempDispositivos.Numero;

      L     #VarTempDispositivos.Numero;  // Comprobar el numero de Llave
      L     1;  // No menor de 1
      <I;  // No es correcto
      JC    Final_EventoRecibido_CSTA;
      L     #VarTempDispositivos.Numero;
      L     "CTE_MaxDispositivosLlave";  // No meyor que el parametro
      >I;  // No es correcto
      JC    Final_EventoRecibido_CSTA;


///////////////////////////////////////////////////////////////////////////////
// --- Guardar el Cambio de Estado Recibido

      SET;
      S     "DB839_DispositivosVarios".DispoLlave[#VarTempDispositivos.Numero].Habilitado;  // Por defecto DesHabilitado

      L     #AtributosDeDispositivos.Habilitado;
      L     2001;  // Nuevo estado - Habilitado SI ?
      ==I;
      JC    HabilitadaLlave_EventoRecibido_CSTA;

      SET;
      R     "DB839_DispositivosVarios".DispoLlave[#VarTempDispositivos.Numero].Habilitado;

HabilitadaLlave_EventoRecibido_CSTA:NOP   0;

      SET;
      S     "DB839_DispositivosVarios".DispoLlave[#VarTempDispositivos.Numero].RefrescoDatos;  // Peticion de Refresco de datos


///////////////////////////////////////////////////////////////////////////////
// Finalizar
      JU    Final_EventoRecibido_CSTA;



NETWORK
TITLE = ---- Accion del Evento --> Notificacion de cambio de Estado de Seta
///////////////////////////////////////////////////////////////////////////////
///////////////////////////////////////////////////////////////////////////////
///////////////////////////////////////////////////////////////////////////////
// --- Tipo Seta
DispositivosSeta_EventoRecibido_CSTA:NOP   0;


///////////////////////////////////////////////////////////////////////////////
// --- Comprobacion del Numero de Dispositivo
      L     #AtributosDeDispositivos.Numero;  // Ver que Seta es
      L     "CTE_OffsetMesa";
      -I;
      T     #VarTempDispositivos.Numero;

      L     #VarTempDispositivos.Numero;  // Comprobar el numero de Seta
      L     1;  // No menor de 1
      <I;  // No es correcto
      JC    Final_EventoRecibido_CSTA;
      L     #VarTempDispositivos.Numero;
      L     "CTE_MaxDispositivosSeta";  // No meyor que el parametro
      >I;  // No es correcto
      JC    Final_EventoRecibido_CSTA;


///////////////////////////////////////////////////////////////////////////////
// --- Guardar el Cambio de Estado Recibido

      SET;
      S     "DB839_DispositivosVarios".DispoSeta[#VarTempDispositivos.Numero].Habilitado;  // Por defecto DesHabilitado

      L     #AtributosDeDispositivos.Habilitado;
      L     2001;  // Nuevo estado - Habilitado SI ?
      ==I;
      JC    HabilitadaSeta_EventoRecibido_CSTA;

      SET;
      R     "DB839_DispositivosVarios".DispoSeta[#VarTempDispositivos.Numero].Habilitado;

HabilitadaSeta_EventoRecibido_CSTA:NOP   0;

      SET;
      S     "DB839_DispositivosVarios".DispoSeta[#VarTempDispositivos.Numero].RefrescoDatos;  // Peticion de Refresco de datos


///////////////////////////////////////////////////////////////////////////////
// Finalizar
      JU    Final_EventoRecibido_CSTA;



NETWORK
TITLE = ---- Accion del Evento --> Notificacion de cambio de Estado de Barrera
///////////////////////////////////////////////////////////////////////////////
///////////////////////////////////////////////////////////////////////////////
///////////////////////////////////////////////////////////////////////////////
// --- Tipo Barrera
DispositivosBarrera_EventoRecibido_CSTA:NOP   0;


///////////////////////////////////////////////////////////////////////////////
// --- Comprobacion del Numero de Dispositivo
      L     #AtributosDeDispositivos.Numero;  // Ver que Barrera es
      L     "CTE_OffsetMesa";
      -I;
      T     #VarTempDispositivos.Numero;

      L     #VarTempDispositivos.Numero;  // Comprobar el numero de Barrera
      L     1;  // No menor de 1
      <I;  // No es correcto
      JC    Final_EventoRecibido_CSTA;
      L     #VarTempDispositivos.Numero;
      L     "CTE_MaxDispositivosBarrera";  // No meyor que el parametro
      >I;  // No es correcto
      JC    Final_EventoRecibido_CSTA;


///////////////////////////////////////////////////////////////////////////////
// --- Guardar el Cambio de Estado Recibido

      SET;
      S     "DB839_DispositivosVarios".DispoBarrera[#VarTempDispositivos.Numero].Habilitado;  // Por defecto DesHabilitado

      L     #AtributosDeDispositivos.Habilitado;
      L     2001;  // Nuevo estado - Habilitado SI ?
      ==I;
      JC    HabilitadaBarrera_EventoRecibido_CSTA;

      SET;
      R     "DB839_DispositivosVarios".DispoBarrera[#VarTempDispositivos.Numero].Habilitado;

HabilitadaBarrera_EventoRecibido_CSTA:NOP   0;

      SET;
      S     "DB839_DispositivosVarios".DispoBarrera[#VarTempDispositivos.Numero].RefrescoDatos;  // Peticion de Refresco de datos


///////////////////////////////////////////////////////////////////////////////
// Finalizar
      JU    Final_EventoRecibido_CSTA;



NETWORK
TITLE = ---- Accion del Evento --> Notificacion de cambio de Estado de Puerta
///////////////////////////////////////////////////////////////////////////////
///////////////////////////////////////////////////////////////////////////////
///////////////////////////////////////////////////////////////////////////////
// --- Tipo Puerta
DispositivosPuerta_EventoRecibido_CSTA:NOP   0;


///////////////////////////////////////////////////////////////////////////////
// --- Comprobacion del Numero de Dispositivo
      L     #AtributosDeDispositivos.Numero;  // Ver que Puerta es
      L     "CTE_OffsetMesa";
      -I;
      T     #VarTempDispositivos.Numero;

      L     #VarTempDispositivos.Numero;  // Comprobar el numero de Puerta
      L     1;  // No menor de 1
      <I;  // No es correcto
      JC    Final_EventoRecibido_CSTA;
      L     #VarTempDispositivos.Numero;
      L     "CTE_MaxDispositivosPuerta";  // No meyor que el parametro
      >I;  // No es correcto
      JC    Final_EventoRecibido_CSTA;


///////////////////////////////////////////////////////////////////////////////
// --- Guardar el Cambio de Estado Recibido

      SET;
      S     "DB839_DispositivosVarios".DispoPuerta[#VarTempDispositivos.Numero].Habilitado;  // Por defecto DesHabilitado

      L     #AtributosDeDispositivos.Habilitado;
      L     2001;  // Nuevo estado - Habilitado SI ?
      ==I;
      JC    HabilitadaPuerta_EventoRecibido_CSTA;

      SET;
      R     "DB839_DispositivosVarios".DispoPuerta[#VarTempDispositivos.Numero].Habilitado;

HabilitadaPuerta_EventoRecibido_CSTA:NOP   0;

      SET;
      S     "DB839_DispositivosVarios".DispoPuerta[#VarTempDispositivos.Numero].RefrescoDatos;  // Peticion de Refresco de datos


///////////////////////////////////////////////////////////////////////////////
// Finalizar
      JU    Final_EventoRecibido_CSTA;



NETWORK
TITLE = ---- Accion del Evento --> Notificacion de cambio de Estado de Linea de Potencia
///////////////////////////////////////////////////////////////////////////////
///////////////////////////////////////////////////////////////////////////////
///////////////////////////////////////////////////////////////////////////////
// --- Tipo Linea de Potencia
DispositivosLineaPotencia_EventoRecibido_CSTA:NOP   0;


///////////////////////////////////////////////////////////////////////////////
// --- Comprobacion del Numero de Dispositivo
      L     #AtributosDeDispositivos.Numero;  // Ver que Linea de Potencia es
      L     "CTE_OffsetMesa";
      -I;
      T     #VarTempDispositivos.Numero;

      L     #VarTempDispositivos.Numero;  // Comprobar el numero de Linea de Potencia
      L     1;  // No menor de 1
      <I;  // No es correcto
      JC    Final_EventoRecibido_CSTA;
      L     #VarTempDispositivos.Numero;
      L     "CTE_MaxDispositivosLlave";  // No meyor que el parametro
      >I;  // No es correcto
      JC    Final_EventoRecibido_CSTA;


///////////////////////////////////////////////////////////////////////////////
// --- Guardar el Cambio de Estado Recibido

      SET;
      S     "DB839_DispositivosVarios".DispoLineaPotencia[#VarTempDispositivos.Numero].Habilitado;  // Por defecto DesHabilitado

      L     #AtributosDeDispositivos.Habilitado;
      L     2001;  // Nuevo estado - Habilitado SI ?
      ==I;
      JC    HabilitadaLineaPotencia_EventoRecibido_CSTA;

      SET;
      R     "DB839_DispositivosVarios".DispoLineaPotencia[#VarTempDispositivos.Numero].Habilitado;

HabilitadaLineaPotencia_EventoRecibido_CSTA:NOP   0;

      SET;
      S     "DB839_DispositivosVarios".DispoLineaPotencia[#VarTempDispositivos.Numero].RefrescoDatos;  // Peticion de Refresco de datos


///////////////////////////////////////////////////////////////////////////////
// Finalizar
      JU    Final_EventoRecibido_CSTA;



NETWORK
TITLE = ---- Final
///////////////////////////////////////////////////////////////////////////////
///////////////////////////////////////////////////////////////////////////////
///////////////////////////////////////////////////////////////////////////////
// Se acabo el evento
Final_EventoRecibido_CSTA:NOP   0;
      L     #P_Eventos;  // Recupero por donde voy en la lista de eventos
      LAR2;
      JU    FinBucle_EventosRecibidos;  // Regreso a buscar el siguiente evento



NETWORK
TITLE = Evento ¿ST? - Peticion de Refresco de los dispositivos
// - Inicializa variables de los atributos del Evento
// - Buscar Atributos o Final del Evento
// - Guardar datos del Evento
//   - Si tiene Tipo y Numero
//   - Si solo Tipo
//   - Si son todos
GuardarDatos_EventoRecibido_Refresco_ST:NOP   0;

/////////////////////////////////////////////////////////////////////////
/////////////////////////////////////////////////////////////////////////
/////////////////////////////////////////////////////////////////////////
// --- Guardar Datos del Evento Recibido
/////////////////////////////////////////////////////////////////////////
/////////////////////////////////////////////////////////////////////////
/////////////////////////////////////////////////////////////////////////
// --- Distribucion por tipo

      SET;  // Dispositivo CCPIF
      L     #AtributosDeDispositivos.Tipo;
      L     50;
      ==I;
      JC    DispositivoCCPIF_EventoRecibido_RefrescoDispositivo;

      SET;  // Dispositivo CBOX
      L     #AtributosDeDispositivos.Tipo;
      L     40;
      ==I;
      JC    DispositivoCBOX_EventoRecibido_RefrescoDispositivo;

      SET;  // Dispositivo Mesa
      L     #AtributosDeDispositivos.Tipo;
      L     60;
      ==I;
      JC    DispositivoMesa_EventoRecibido_RefrescoDispositivo;


///////////////////////////////////////////////////////////////////////////////
///////////////////////////////////////////////////////////////////////////////
///////////////////////////////////////////////////////////////////////////////

      SET;  // Dispositivos Baliza
      L     #AtributosDeDispositivos.Tipo;
      L     1000;
      ==I;
      JC    DispositivoBaliza_EventoRecibido_RefrescoDispositivo;

      SET;  // Dispositivos Llave
      L     #AtributosDeDispositivos.Tipo;
      L     1001;
      ==I;
      JC    DispositivoLlave_EventoRecibido_RefrescoDispositivo;

      SET;  // Dispositivos Seta
      L     #AtributosDeDispositivos.Tipo;
      L     1002;
      ==I;
      JC    DispositivoSeta_EventoRecibido_RefrescoDispositivo;

      SET;  // Dispositivos Barrera
      L     #AtributosDeDispositivos.Tipo;
      L     1003;
      ==I;
      JC    DispositivoBarrera_EventoRecibido_RefrescoDispositivo;

      SET;  // Dispositivos Puerta
      L     #AtributosDeDispositivos.Tipo;
      L     1004;
      ==I;
      JC    DispositivoPuerta_EventoRecibido_RefrescoDispositivo;

      SET;  // Dispositivos Linea de Potencia
      L     #AtributosDeDispositivos.Tipo;
      L     1005;
      ==I;
      JC    DispositivoLineaPotencia_EventoRecibido_RefrescoDispositivo;


///////////////////////////////////////////////////////////////////////////////
///////////////////////////////////////////////////////////////////////////////
///////////////////////////////////////////////////////////////////////////////
// Dispositivo Maquina De 70 ... 99
      SET;
      A(;
      L     #AtributosDeDispositivos.Tipo;
      L     70;
      >=I;
      );
      A(;
      L     #AtributosDeDispositivos.Tipo;
      L     99;
      <=I;
      );
      JC    DispositivoMaquina_EventoRecibido_RefrescoDispositivo;


///////////////////////////////////////////////////////////////////////////////
///////////////////////////////////////////////////////////////////////////////
///////////////////////////////////////////////////////////////////////////////
// --- Todos los dipositivos -> Por defecto
      JU    DispositivosTodos_EventoRecibido_RefrescoDispositivo;



NETWORK
TITLE = ---- Accion del Evento --> Peticion de Refresco del Dispositivo CCPIF
///////////////////////////////////////////////////////////////////////////////
///////////////////////////////////////////////////////////////////////////////
///////////////////////////////////////////////////////////////////////////////
// Dispositivos tipo CCPIF
DispositivoCCPIF_EventoRecibido_RefrescoDispositivo:NOP   0;
      SET;
      L     #AtributosDeDispositivos.Numero;  // No se envia Numero CCPIF
      L     0;  // Son todos los CCPIF's (Solo uno)
      ==I;
      JC    RefrescoDipositivoCCPIF_RefrescoDispositivo_EventosRecibidos;

      L     #AtributosDeDispositivos.Numero;  // Comprobacion del numero de CCPIF
      L     "CTE_OffsetCCPIF";
      -I;
      L     1;
      <>I;  // Numero de CCPIF incorrecto
      JC    Final_EventoRecibido_RefrescoDispositivo;


///////////////////////////////////////////////////////////////////////////////
// Activar Refresco del Dispositivo
RefrescoDipositivoCCPIF_RefrescoDispositivo_EventosRecibidos:NOP   0;

      L     250;  // 250 - Recibido Evento de Refresco de Datos del Dispositivo
      T     "DB830_Dispositivos".Dispositivos[0].EstadoRecepcionEvento;


///////////////////////////////////////////////////////////////////////////////
// Finalizar
      JU    Final_EventoRecibido_RefrescoDispositivo;



NETWORK
TITLE = ---- Accion del Evento --> Peticion de Refresco del Dispositivo CBOX
///////////////////////////////////////////////////////////////////////////////
///////////////////////////////////////////////////////////////////////////////
///////////////////////////////////////////////////////////////////////////////
// --- Dispositivos tipo CBOX, uno determinado o todos
DispositivoCBOX_EventoRecibido_RefrescoDispositivo:NOP   0;
      SET;
      L     #AtributosDeDispositivos.Numero;  // Mirar si hay numero de CBOX
      L     0;  // Son todos los CBOX's
      ==I;
      JC    DispositivosTodosCBOX_EventoRecibido_RefrescoDispositivo;


///////////////////////////////////////////////////////////////////////////////
// --- Es Un CBOX Determinado
      JU    DispositivoUnCBOX_EventoRecibido_RefrescoDispositivo;



NETWORK
TITLE = ---- ---- De un CBOX
///////////////////////////////////////////////////////////////////////////////
///////////////////////////////////////////////////////////////////////////////
///////////////////////////////////////////////////////////////////////////////
// --- Un CBOX determinado
DispositivoUnCBOX_EventoRecibido_RefrescoDispositivo:NOP   0;


///////////////////////////////////////////////////////////////////////////////
// --- Comprobacion del numero de CCPIF
      L     #AtributosDeDispositivos.Numero;
      L     100;
      /I;
      L     "CTE_OffsetCCPIF";
      -I;
      L     1;
      <>I;  // Numero de CCPIF incorrecto
      JC    Final_EventoRecibido_RefrescoDispositivo;

      L     #AtributosDeDispositivos.Numero;  // Calculo del numero de CBOX
      L     100;
      MOD;  // Var verlo en la DB_Dispositivos
      T     #VarTempDispositivos.Numero;

      L     #VarTempDispositivos.Numero;  // Comprobacion del numero de CBOX
      L     1;  // Es menor de 1
      <I;  // No es correcto el numero de CBOX
      JC    Final_EventoRecibido_RefrescoDispositivo;
      L     #VarTempDispositivos.Numero;
      L     "CTE_MaxDispositivos";  // Si es mayor que el parametro
      >I;  // No es correcto el nuemro de CBOX
      JC    Final_EventoRecibido_RefrescoDispositivo;


///////////////////////////////////////////////////////////////////////////////
// --- Activar Refresco del Dispositivo
      L     250;  // 250 - Recibido Evento de Refresco de Datos del Dispositivo
      T     "DB830_Dispositivos".Dispositivos[#VarTempDispositivos.Numero].EstadoRecepcionEvento;


///////////////////////////////////////////////////////////////////////////////
// --- Finalizar
      JU    Final_EventoRecibido_RefrescoDispositivo;



NETWORK
TITLE = ---- ---- De Todos los CBOX
///////////////////////////////////////////////////////////////////////////////
///////////////////////////////////////////////////////////////////////////////
///////////////////////////////////////////////////////////////////////////////
// --- Son todos los CBOX
DispositivosTodosCBOX_EventoRecibido_RefrescoDispositivo:NOP   0;
      L     1;
      T     #IndiceCBOX;


///////////////////////////////////////////////////////////////////////////////
///////////////////////////////////////////////////////////////////////////////
///////////////////////////////////////////////////////////////////////////////
// --- Recorrer todo los dispositivos
BucleDispositivosTodosCBOX_EventoRecibido_RefrescoDispositivo:NOP   0;

// Mirar si Pertenece al JDT
      SET;
      X     "DB855_DefinicionDispositivos".Dispositivos[#IndiceCBOX].EventosDelJdT02;
      XN    #JDT02_Activo;
      =     #DispositivoDeJDT02;

      SET;
      AN    #DispositivoDeJDT02;
      JC    ContinuarBucleDispositivosTodosCBOX_EventoRecibido_RefrescoDispositivo;


///////////////////////////////////////////////////////////////////////////////
// Activar Refresco del Dispositivo
      L     250;  // 250 - Recibido Evento de Refresco de Datos del Dispositivo
      T     "DB830_Dispositivos".Dispositivos[#IndiceCBOX].EstadoRecepcionEvento;


///////////////////////////////////////////////////////////////////////////////
// Ir hacia el siguiente CBOX
ContinuarBucleDispositivosTodosCBOX_EventoRecibido_RefrescoDispositivo:NOP   0;
      L     #IndiceCBOX;  // Incremento al siguiente CBOX
      L     1;
      +I;
      T     #IndiceCBOX;

      L     #IndiceCBOX;
      L     "CTE_MaxDispositivos";
      >I;  // Finalizar
      JC    Final_EventoRecibido_RefrescoDispositivo;

///////////////////////////////////////////////////////////////////////////////
      JU    BucleDispositivosTodosCBOX_EventoRecibido_RefrescoDispositivo;



NETWORK
TITLE = ---- Accion del Evento --> Peticion de Refresco del Dispositivo Mesa
///////////////////////////////////////////////////////////////////////////////
///////////////////////////////////////////////////////////////////////////////
///////////////////////////////////////////////////////////////////////////////
// --- Dispositivos tipo Mesa, uno determinado o todos
DispositivoMesa_EventoRecibido_RefrescoDispositivo:NOP   0;
      SET;
      L     #AtributosDeDispositivos.Numero;  // Mirar si hay numero de Mesas
      L     0;  // Son todos los Mesas
      ==I;
      JC    DispositivosTodosMesa_EventoRecibido_RefrescoDispositivo;


///////////////////////////////////////////////////////////////////////////////
// --- Es Una Mesa Determinada
      JU    DispositivosUnaMesa_EventoRecibido_RefrescoDispositivo;




NETWORK
TITLE = ---- ---- De una Mesa
///////////////////////////////////////////////////////////////////////////////
///////////////////////////////////////////////////////////////////////////////
///////////////////////////////////////////////////////////////////////////////
// --- Una Mesa determinada
DispositivosUnaMesa_EventoRecibido_RefrescoDispositivo:NOP   0;

      L     #AtributosDeDispositivos.Numero;  // Ver que mesa es
      L     "CTE_OffsetMesa";
      -I;
      T     #VarTempDispositivos.Numero;

      L     #VarTempDispositivos.Numero;  // Comprobar el numero de mesa
      L     1;  // No menor de 1
      <I;  // No es correcto
      JC    Final_EventoRecibido_RefrescoDispositivo;
      L     #VarTempDispositivos.Numero;
      L     "CTE_MaxMesas";  // No meyor que el parametro
      >I;  // No es correcto
      JC    Final_EventoRecibido_RefrescoDispositivo;


///////////////////////////////////////////////////////////////////////////////
// --- Activar Refresco del Dispositivo
      L     250;  // 250 - Recibido Evento de Refresco de Datos del Dispositivo
      T     "DB831_Mesas".Mesas[#VarTempDispositivos.Numero].EstadoRecepcionEvento;


///////////////////////////////////////////////////////////////////////////////
// --- Finalizar
      JU    Final_EventoRecibido_RefrescoDispositivo;



NETWORK
TITLE = ---- ---- De Todas las Mesas
///////////////////////////////////////////////////////////////////////////////
///////////////////////////////////////////////////////////////////////////////
///////////////////////////////////////////////////////////////////////////////
// --- Todas las Mesas
DispositivosTodosMesa_EventoRecibido_RefrescoDispositivo:NOP   0;
      L     1;
      T     #IndiceMesa;


///////////////////////////////////////////////////////////////////////////////
///////////////////////////////////////////////////////////////////////////////
///////////////////////////////////////////////////////////////////////////////
// Recorrer todo los dispositivos
BucleDispositivosTodosMesa_EventoRecibido_RefrescoDispositivo:NOP   0;


///////////////////////////////////////////////////////////////////////////////
// Mirar si esta definido como mesa de Tracking y TL
      SET;
      AN    "DB850_DefinicionMesas".Mesa[#IndiceMesa].ConfigMesa.MesaPaso;
      AN    "DB850_DefinicionMesas".Mesa[#IndiceMesa].ConfigMesa.MesaCruce;
      AN    "DB850_DefinicionMesas".Mesa[#IndiceMesa].ConfigMesa.MesaMultiplesDestinos;
      AN    "DB850_DefinicionMesas".Mesa[#IndiceMesa].ConfigMesa.MesaTL;
      JC    ContinuarBucleDispositivosTodosMesa_EventoRecibido_RefrescoDispositivo;


///////////////////////////////////////////////////////////////////////////////
/// Mirar Si pertenece al JDT
      SET;
      X     "DB850_DefinicionMesas".Mesa[#IndiceMesa].ConfigMesa.MesaDeJDT02;  // JDT01 ?
      XN    #JDT02_Activo;
      =     #DispositivoDeJDT02;

      SET;
      AN    #DispositivoDeJDT02;
      JC    ContinuarBucleDispositivosTodosMesa_EventoRecibido_RefrescoDispositivo;


///////////////////////////////////////////////////////////////////////////////
// Activar Refresco del Dispositivo
      L     250;  // 250 - Recibido Evento de Refresco de Datos del Dispositivo
      T     "DB831_Mesas".Mesas[#IndiceMesa].EstadoRecepcionEvento;


///////////////////////////////////////////////////////////////////////////////
ContinuarBucleDispositivosTodosMesa_EventoRecibido_RefrescoDispositivo:NOP   0;
      L     #IndiceMesa;  // Incremento al siguiente Mesa
      L     1;
      +I;
      T     #IndiceMesa;

      L     #IndiceMesa;
      L     "CTE_MaxMesas";
      >I;  // Finalizar
      JC    Final_EventoRecibido_RefrescoDispositivo;


///////////////////////////////////////////////////////////////////////////////
// -- Ir hacia el siguiente Mesa
      JU    BucleDispositivosTodosMesa_EventoRecibido_RefrescoDispositivo;



NETWORK
TITLE = ---- Accion del Evento --> Peticion de Refresco del Dispositivo Maquinas
///////////////////////////////////////////////////////////////////////////////
///////////////////////////////////////////////////////////////////////////////
///////////////////////////////////////////////////////////////////////////////
// Dispositivos tipo Maquina uno determinado o todos
DispositivoMaquina_EventoRecibido_RefrescoDispositivo:NOP   0;
      SET;
      L     #AtributosDeDispositivos.Numero;  // Mirar si hay numero de maquina
      L     0;  // Son todos los CBOX's
      ==I;
      JC    DispositivosTodosMaquina_EventoRecibido_RefrescoDispositivo;


///////////////////////////////////////////////////////////////////////////////
// --- Es Una Maquina Determinada
      JU    DispositivosUnaMaquina_EventoRecibido_RefrescoDispositivo;



NETWORK
TITLE = ---- ---- De una Maquina
///////////////////////////////////////////////////////////////////////////////
///////////////////////////////////////////////////////////////////////////////
///////////////////////////////////////////////////////////////////////////////
// --- Maquina  determinada
DispositivosUnaMaquina_EventoRecibido_RefrescoDispositivo:NOP   0;

      L     #AtributosDeDispositivos.Numero;  // Ver que maquina es
      L     "CTE_OffsetMesa";
      -I;
      T     #VarTempDispositivos.Numero;

      L     #VarTempDispositivos.Numero;  // Comprobar el numero de maquina
      L     1;  // No menor de 1
      <I;  // No es correcto
      JC    Final_EventoRecibido_RefrescoDispositivo;
      L     #VarTempDispositivos.Numero;
      L     "CTE_MaxMesas";  // No meyor que el parametro
      >I;  // No es correcto
      JC    Final_EventoRecibido_RefrescoDispositivo;


///////////////////////////////////////////////////////////////////////////////
// --- Activar Refresco del Dispositivo
      L     250;  // 250 - Recibido Evento de Refresco de Datos del Dispositivo
      T     "DB832_Maquinas".Maquinas[#VarTempDispositivos.Numero].EstadoRecepcionEvento;


///////////////////////////////////////////////////////////////////////////////
// --- Finalizar
      JU    Final_EventoRecibido_RefrescoDispositivo;



NETWORK
TITLE = ---- ---- De Todas las Maquinas
///////////////////////////////////////////////////////////////////////////////
///////////////////////////////////////////////////////////////////////////////
///////////////////////////////////////////////////////////////////////////////
// --- Todas las Maquinas
DispositivosTodosMaquina_EventoRecibido_RefrescoDispositivo:NOP   0;
      L     1;
      T     #IndiceMaquina;


///////////////////////////////////////////////////////////////////////////////
///////////////////////////////////////////////////////////////////////////////
///////////////////////////////////////////////////////////////////////////////
BucleDispositivosTodosMaquina_EventoRecibido_RefrescoDispositivo:NOP   0;


///////////////////////////////////////////////////////////////////////////////
// --- Mirar si esta definido como mesa de Tracking y TL
      SET;
      AN    "DB850_DefinicionMesas".Mesa[#IndiceMaquina].ConfigMesa.MesaPaso;
      AN    "DB850_DefinicionMesas".Mesa[#IndiceMaquina].ConfigMesa.MesaCruce;
      AN    "DB850_DefinicionMesas".Mesa[#IndiceMaquina].ConfigMesa.MesaMultiplesDestinos;
      AN    "DB850_DefinicionMesas".Mesa[#IndiceMaquina].ConfigMesa.MesaTL;
      JC    ContinuarBucleDispositivosTodosMaquina_EventoRecibido_RefrescoDispositivo;


///////////////////////////////////////////////////////////////////////////////
/// Mirar Si hay maquina
      SET;
      AN    "DB850_DefinicionMesas".Mesa[#IndiceMaquina].ConfigMesa.MaquinaEnMesa;  // Maquina ?
      JC    ContinuarBucleDispositivosTodosMaquina_EventoRecibido_RefrescoDispositivo;


///////////////////////////////////////////////////////////////////////////////
/// --- Mirar Si pertenece al JDT
      SET;
      X     "DB850_DefinicionMesas".Mesa[#IndiceMaquina].ConfigMesa.MesaDeJDT02;  // JDT01 ?
      XN    #JDT02_Activo;
      =     #DispositivoDeJDT02;

      SET;
      AN    #DispositivoDeJDT02;
      JC    ContinuarBucleDispositivosTodosMaquina_EventoRecibido_RefrescoDispositivo;


///////////////////////////////////////////////////////////////////////////////
// --- Activar Refresco del Dispositivo
      L     250;  // 250 - Recibido Evento de Refresco de Datos del Dispositivo
      T     "DB832_Maquinas".Maquinas[#IndiceMaquina].EstadoRecepcionEvento;


///////////////////////////////////////////////////////////////////////////////
ContinuarBucleDispositivosTodosMaquina_EventoRecibido_RefrescoDispositivo:NOP   0;
      L     #IndiceMaquina;  // Incremento al siguiente Maquina
      L     1;
      +I;
      T     #IndiceMaquina;

      L     #IndiceMaquina;
      L     "CTE_MaxMesas";
      >I;  // Finalizar
      JC    Final_EventoRecibido_RefrescoDispositivo;


///////////////////////////////////////////////////////////////////////////////
// --- Ir hacia el siguiente Maquina
      JU    BucleDispositivosTodosMaquina_EventoRecibido_RefrescoDispositivo;



NETWORK
TITLE = ---- Accion del Evento --> Peticion de Refresco del Dispositivo Baliza
///////////////////////////////////////////////////////////////////////////////
///////////////////////////////////////////////////////////////////////////////
///////////////////////////////////////////////////////////////////////////////
// Dispositivos tipo Baliza uno determinado o todos
DispositivoBaliza_EventoRecibido_RefrescoDispositivo:NOP   0;
      SET;
      L     #AtributosDeDispositivos.Numero;  // Mirar si hay numero de maquina
      L     0;  // Son todos las Balizas
      ==I;
      JC    DispositivosTodosBaliza_EventoRecibido_RefrescoDispositivo;


///////////////////////////////////////////////////////////////////////////////
// --- Es Una Maquina Determinada
      JU    DispositivosUnaBaliza_EventoRecibido_RefrescoDispositivo;



NETWORK
TITLE = ---- ---- De una Baliza
///////////////////////////////////////////////////////////////////////////////
///////////////////////////////////////////////////////////////////////////////
///////////////////////////////////////////////////////////////////////////////
// --- Una Baliza determinada
DispositivosUnaBaliza_EventoRecibido_RefrescoDispositivo:NOP   0;

      L     #AtributosDeDispositivos.Numero;  // Ver que Baliza es
      L     "CTE_OffsetMesa";
      -I;
      T     #VarTempDispositivos.Numero;

      L     #VarTempDispositivos.Numero;  // Comprobar el numero de Baliza
      L     1;  // No menor de 1
      <I;  // No es correcto
      JC    Final_EventoRecibido_RefrescoDispositivo;
      L     #VarTempDispositivos.Numero;
      L     "CTE_MaxDispositivosBaliza";  // No meyor que el parametro
      >I;  // No es correcto
      JC    Final_EventoRecibido_RefrescoDispositivo;


///////////////////////////////////////////////////////////////////////////////
// --- Activar Refresco del Dispositivo
///////////////////////////////////////////////////////////////////////////////
// Activar Refresco del Dispositivo
      SET;
      S     "DB839_DispositivosVarios".DispoBaliza[#VarTempDispositivos.Numero].RefrescoDatos;


///////////////////////////////////////////////////////////////////////////////
// --- Finalizar
      JU    Final_EventoRecibido_RefrescoDispositivo;



NETWORK
TITLE = ---- ---- De Todas las Balizas
////////////////////////////////////////////////////////////////////////////
////////////////////////////////////////////////////////////////////////////
////////////////////////////////////////////////////////////////////////////
// --- Peticion de Todos los dispositivos BALIZA
DispositivosTodosBaliza_EventoRecibido_RefrescoDispositivo:NOP   0;
      L     1;
      T     #IndiceDispositivosVarios;


////////////////////////////////////////////////////////////////////////////
////////////////////////////////////////////////////////////////////////////
////////////////////////////////////////////////////////////////////////////
BucleBaliza_EventoRecibido_RefrescoDispositivo:NOP   0;


///////////////////////////////////////////////////////////////////////////////
// Activar Refresco del Dispositivo
      SET;
      S     "DB839_DispositivosVarios".DispoBaliza[#IndiceDispositivosVarios].RefrescoDatos;

////////////////////////////////////////////////////////////////////////////
      L     #IndiceDispositivosVarios;  // Siguiente Dispositivo
      L     1;
      +I;
      T     #IndiceDispositivosVarios;

      L     #IndiceDispositivosVarios;
      L     "CTE_MaxDispositivosBaliza";
      >I;  // Ha superado el maximo ??
      JC    FinBucleBaliza_EventoRecibido_RefrescoDispositivo;

      JU    BucleBaliza_EventoRecibido_RefrescoDispositivo;  // Continuar en el Bucle


////////////////////////////////////////////////////////////////////////////
////////////////////////////////////////////////////////////////////////////
////////////////////////////////////////////////////////////////////////////
FinBucleBaliza_EventoRecibido_RefrescoDispositivo:NOP   0;
      JU    Final_EventoRecibido_RefrescoDispositivo;


NETWORK
TITLE = ---- Accion del Evento --> Peticion de Refresco del Dispositivo Llave
///////////////////////////////////////////////////////////////////////////////
///////////////////////////////////////////////////////////////////////////////
///////////////////////////////////////////////////////////////////////////////
// Dispositivos tipo Llave uno determinado o todos
DispositivoLlave_EventoRecibido_RefrescoDispositivo:NOP   0;
      SET;
      L     #AtributosDeDispositivos.Numero;  // Mirar si hay numero de maquina
      L     0;  // Son todos las Llaves
      ==I;
      JC    DispositivosTodosLlave_EventoRecibido_RefrescoDispositivo;


///////////////////////////////////////////////////////////////////////////////
// --- Es Una Maquina Determinada
      JU    DispositivosUnaLlave_EventoRecibido_RefrescoDispositivo;



NETWORK
TITLE = ---- ---- De una Llave
///////////////////////////////////////////////////////////////////////////////
///////////////////////////////////////////////////////////////////////////////
///////////////////////////////////////////////////////////////////////////////
// --- Una Llave determinada
DispositivosUnaLlave_EventoRecibido_RefrescoDispositivo:NOP   0;

      L     #AtributosDeDispositivos.Numero;  // Ver que Llave es
      L     "CTE_OffsetMesa";
      -I;
      T     #VarTempDispositivos.Numero;

      L     #VarTempDispositivos.Numero;  // Comprobar el numero de Llave
      L     1;  // No menor de 1
      <I;  // No es correcto
      JC    Final_EventoRecibido_RefrescoDispositivo;
      L     #VarTempDispositivos.Numero;
      L     "CTE_MaxDispositivosLlave";  // No meyor que el parametro
      >I;  // No es correcto
      JC    Final_EventoRecibido_RefrescoDispositivo;


///////////////////////////////////////////////////////////////////////////////
// --- Activar Refresco del Dispositivo
///////////////////////////////////////////////////////////////////////////////
// Activar Refresco del Dispositivo
      SET;
      S     "DB839_DispositivosVarios".DispoLlave[#VarTempDispositivos.Numero].RefrescoDatos;


///////////////////////////////////////////////////////////////////////////////
// --- Finalizar
      JU    Final_EventoRecibido_RefrescoDispositivo;



NETWORK
TITLE = ---- ---- De Todas las Llaves
////////////////////////////////////////////////////////////////////////////
////////////////////////////////////////////////////////////////////////////
////////////////////////////////////////////////////////////////////////////
// --- Peticion de Todos los dispositivos LLAVE
DispositivosTodosLlave_EventoRecibido_RefrescoDispositivo:NOP   0;
      L     1;
      T     #IndiceDispositivosVarios;


////////////////////////////////////////////////////////////////////////////
////////////////////////////////////////////////////////////////////////////
////////////////////////////////////////////////////////////////////////////
BucleLlave_EventoRecibido_RefrescoDispositivo:NOP   0;


///////////////////////////////////////////////////////////////////////////////
// Activar Refresco del Dispositivo
      SET;
      S     "DB839_DispositivosVarios".DispoLlave[#IndiceDispositivosVarios].RefrescoDatos;
////////////////////////////////////////////////////////////////////////////
      L     #IndiceDispositivosVarios;  // Siguiente Dispositivo
      L     1;
      +I;
      T     #IndiceDispositivosVarios;

      L     #IndiceDispositivosVarios;
      L     "CTE_MaxDispositivosLlave";
      >I;  // Ha superado el maximo ??
      JC    FinBuclellave_EventoRecibido_RefrescoDispositivo;

      JU    BucleLlave_EventoRecibido_RefrescoDispositivo;  // Continuar en el Bucle


////////////////////////////////////////////////////////////////////////////
////////////////////////////////////////////////////////////////////////////
////////////////////////////////////////////////////////////////////////////
FinBuclellave_EventoRecibido_RefrescoDispositivo:NOP   0;
      JU    Final_EventoRecibido_RefrescoDispositivo;


NETWORK
TITLE = ---- Accion del Evento --> Peticion de Refresco del Dispositivo Seta
///////////////////////////////////////////////////////////////////////////////
///////////////////////////////////////////////////////////////////////////////
///////////////////////////////////////////////////////////////////////////////
// Dispositivos tipo Seta uno determinado o todos
DispositivoSeta_EventoRecibido_RefrescoDispositivo:NOP   0;
      SET;
      L     #AtributosDeDispositivos.Numero;  // Mirar si hay numero de maquina
      L     0;  // Son todos las Setas
      ==I;
      JC    DispositivosTodosSeta_EventoRecibido_RefrescoDispositivo;


///////////////////////////////////////////////////////////////////////////////
// --- Es Una Maquina Determinada
      JU    DispositivosUnaSeta_EventoRecibido_RefrescoDispositivo;



NETWORK
TITLE = ---- ---- De una Seta
///////////////////////////////////////////////////////////////////////////////
///////////////////////////////////////////////////////////////////////////////
///////////////////////////////////////////////////////////////////////////////
// --- Una Seta determinada
DispositivosUnaSeta_EventoRecibido_RefrescoDispositivo:NOP   0;

      L     #AtributosDeDispositivos.Numero;  // Ver que Seta es
      L     "CTE_OffsetMesa";
      -I;
      T     #VarTempDispositivos.Numero;

      L     #VarTempDispositivos.Numero;  // Comprobar el numero de Seta
      L     1;  // No menor de 1
      <I;  // No es correcto
      JC    Final_EventoRecibido_RefrescoDispositivo;
      L     #VarTempDispositivos.Numero;
      L     "CTE_MaxDispositivosSeta";  // No meyor que el parametro
      >I;  // No es correcto
      JC    Final_EventoRecibido_RefrescoDispositivo;


///////////////////////////////////////////////////////////////////////////////
// --- Activar Refresco del Dispositivo
///////////////////////////////////////////////////////////////////////////////
// Activar Refresco del Dispositivo
      SET;
      S     "DB839_DispositivosVarios".DispoSeta[#VarTempDispositivos.Numero].RefrescoDatos;


///////////////////////////////////////////////////////////////////////////////
// --- Finalizar
      JU    Final_EventoRecibido_RefrescoDispositivo;



NETWORK
TITLE = ---- ---- De Todas las Setas
////////////////////////////////////////////////////////////////////////////
////////////////////////////////////////////////////////////////////////////
////////////////////////////////////////////////////////////////////////////
// --- Peticion de Todos los dispositivos SETA
DispositivosTodosSeta_EventoRecibido_RefrescoDispositivo:NOP   0;
      L     1;
      T     #IndiceDispositivosVarios;


////////////////////////////////////////////////////////////////////////////
////////////////////////////////////////////////////////////////////////////
////////////////////////////////////////////////////////////////////////////
BucleSeta_EventoRecibido_RefrescoDispositivo:NOP   0;


///////////////////////////////////////////////////////////////////////////////
// Activar Refresco del Dispositivo
      SET;
      S     "DB839_DispositivosVarios".DispoSeta[#IndiceDispositivosVarios].RefrescoDatos;
////////////////////////////////////////////////////////////////////////////
      L     #IndiceDispositivosVarios;  // Siguiente Dispositivo
      L     1;
      +I;
      T     #IndiceDispositivosVarios;

      L     #IndiceDispositivosVarios;
      L     "CTE_MaxDispositivosSeta";
      >I;  // Ha superado el maximo ??
      JC    FinBucleSeta_EventoRecibido_RefrescoDispositivo;

      JU    BucleSeta_EventoRecibido_RefrescoDispositivo;  // Continuar en el Bucle


////////////////////////////////////////////////////////////////////////////
////////////////////////////////////////////////////////////////////////////
////////////////////////////////////////////////////////////////////////////
FinBucleSeta_EventoRecibido_RefrescoDispositivo:NOP   0;
      JU    Final_EventoRecibido_RefrescoDispositivo;


